// NETWORK 4
gvl_axis.fbi_mc_absR(
    Axis := gvl_axis.axisR,
    Execute := gvl_axis.ref_r.Execute,
    Position := gvl_axis.ref_r.Position,
    Velocity := gvl_axis.ref_r.Velocity,
    Acceleration := gvl_axis.ref_r.Acceleration,
    Deceleration := gvl_axis.ref_r.Deceleration,
    Jerk := gvl_axis.ref_r.Jerk,
    BufferMode := gvl_axis.ref_r.BufferMode,
    Options := gvl_axis.ref_r.Options,
    Busy => gvl_axis.ref_r.Busy,
    Active => gvl_axis.ref_r.Active,
    CommandAborted => gvl_axis.ref_r.CommandAborted,
    Error => gvl_axis.ref_r.Error,
    ErrorID => gvl_axis.ref_r.ErrorID); // MC_MoveAbsolute
gvl_axis.ref_r.Done := gvl_axis.fbi_mc_absR.Done;

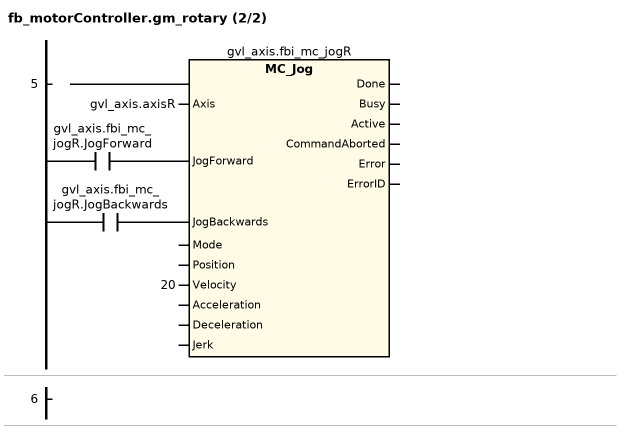
// NETWORK 5
gvl_axis.fbi_mc_jogR(
    Axis := gvl_axis.axisR,
    JogForward := gvl_axis.fbi_mc_jogR.JogForward,
    JogBackwards := gvl_axis.fbi_mc_jogR.JogBackwards,
    Velocity := 20); // MC_Jog

// NETWORK 6
END_ACTION

ACTION motorJog:
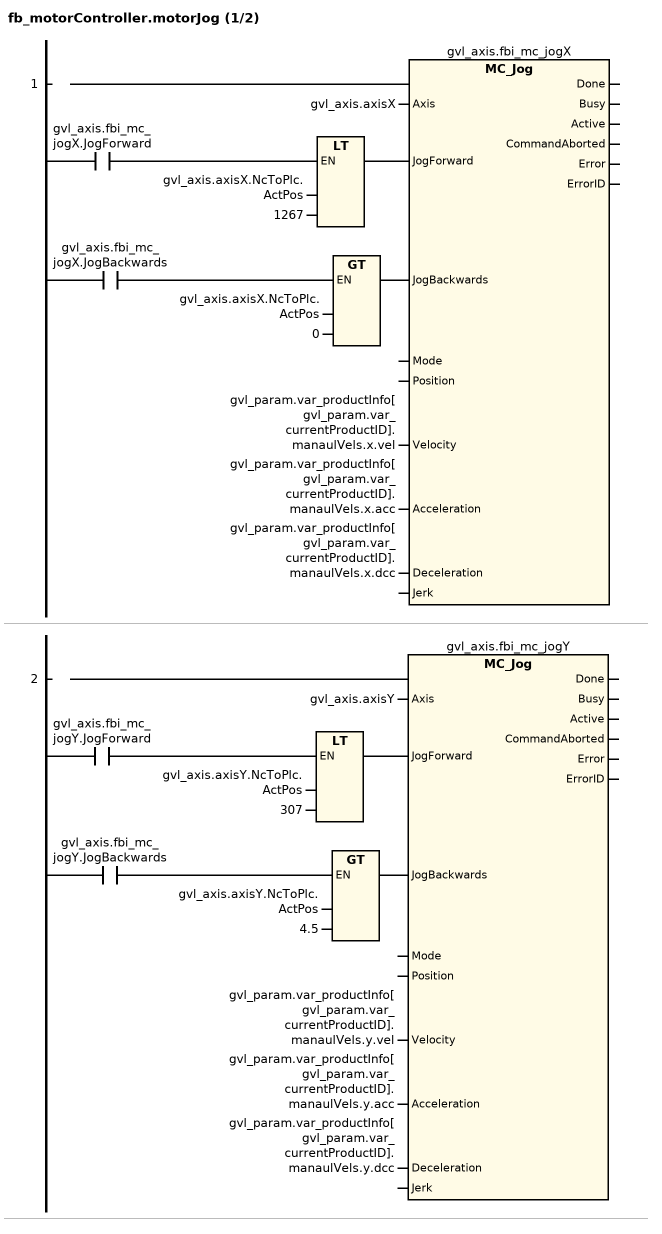
// NETWORK 1
gvl_axis.fbi_mc_jogX(
    Axis := gvl_axis.axisX,
    JogForward := gvl_axis.fbi_mc_jogX.JogForward AND gvl_axis.axisX.NcToPlc.ActPos < 1267,
    JogBackwards := gvl_axis.fbi_mc_jogX.JogBackwards AND gvl_axis.axisX.NcToPlc.ActPos > 0,
    Velocity := gvl_param.var_productInfo[gvl_param.var_currentProductID].manaulVels.x.vel,
    Acceleration := gvl_param.var_productInfo[gvl_param.var_currentProductID].manaulVels.x.acc,
    Deceleration := gvl_param.var_productInfo[gvl_param.var_currentProductID].manaulVels.x.dcc); // MC_Jog

// NETWORK 2
gvl_axis.fbi_mc_jogY(
    Axis := gvl_axis.axisY,
    JogForward := gvl_axis.fbi_mc_jogY.JogForward AND gvl_axis.axisY.NcToPlc.ActPos < 307,
    JogBackwards := gvl_axis.fbi_mc_jogY.JogBackwards AND gvl_axis.axisY.NcToPlc.ActPos > 4.5,
    Velocity := gvl_param.var_productInfo[gvl_param.var_currentProductID].manaulVels.y.vel,
    Acceleration := gvl_param.var_productInfo[gvl_param.var_currentProductID].manaulVels.y.acc,
    Deceleration := gvl_param.var_productInfo[gvl_param.var_currentProductID].manaulVels.y.dcc); // MC_Jog

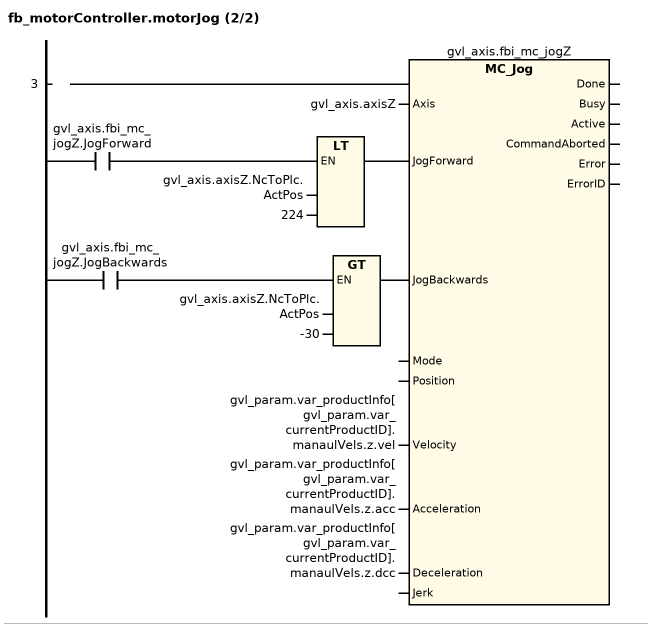
// NETWORK 3
gvl_axis.fbi_mc_jogZ(
    Axis := gvl_axis.axisZ,
    JogForward := gvl_axis.fbi_mc_jogZ.JogForward AND gvl_axis.axisZ.NcToPlc.ActPos < 224,
    JogBackwards := gvl_axis.fbi_mc_jogZ.JogBackwards AND gvl_axis.axisZ.NcToPlc.ActPos > -30,
    Velocity := gvl_param.var_productInfo[gvl_param.var_currentProductID].manaulVels.z.vel,
    Acceleration := gvl_param.var_productInfo[gvl_param.var_currentProductID].manaulVels.z.acc,
    Deceleration := gvl_param.var_productInfo[gvl_param.var_currentProductID].manaulVels.z.dcc); // MC_Jog
END_ACTION

ACTION motorMoveAbs:
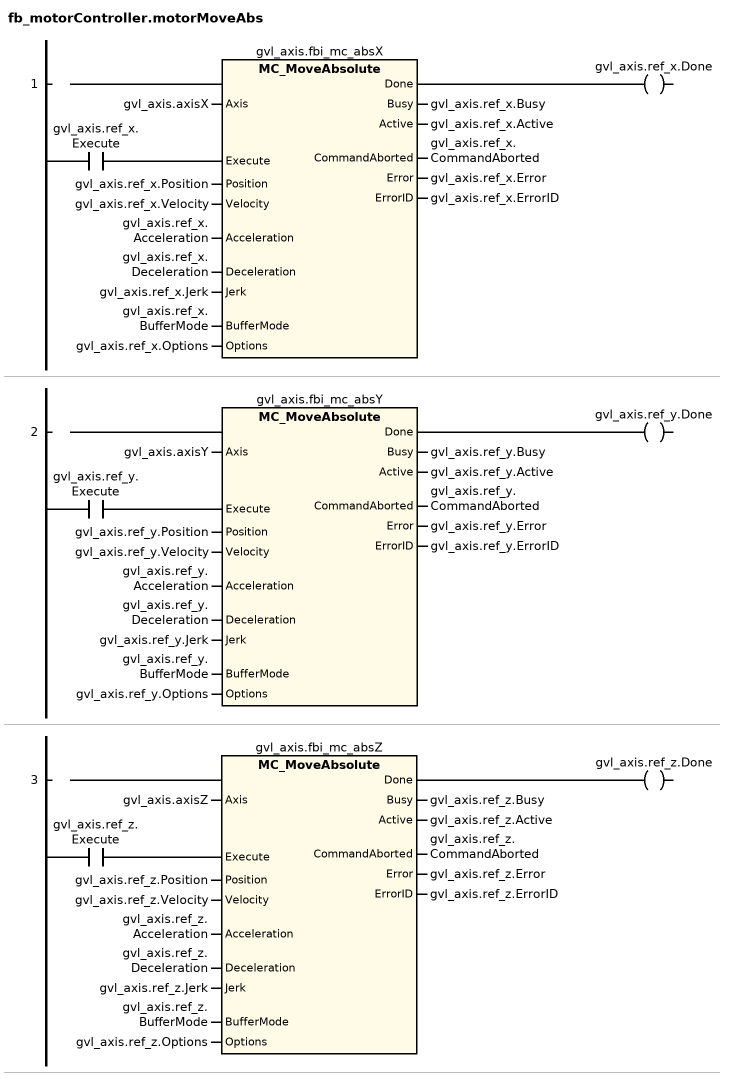
// NETWORK 1
gvl_axis.fbi_mc_absX(
    Axis := gvl_axis.axisX,
    Execute := gvl_axis.ref_x.Execute,
    Position := gvl_axis.ref_x.Position,
    Velocity := gvl_axis.ref_x.Velocity,
    Acceleration := gvl_axis.ref_x.Acceleration,
    Deceleration := gvl_axis.ref_x.Deceleration,
    Jerk := gvl_axis.ref_x.Jerk,
    BufferMode := gvl_axis.ref_x.BufferMode,
    Options := gvl_axis.ref_x.Options,
    Busy => gvl_axis.ref_x.Busy,
    Active => gvl_axis.ref_x.Active,
    CommandAborted => gvl_axis.ref_x.CommandAborted,
    Error => gvl_axis.ref_x.Error,
    ErrorID => gvl_axis.ref_x.ErrorID); // MC_MoveAbsolute
gvl_axis.ref_x.Done := gvl_axis.fbi_mc_absX.Done;

// NETWORK 2
gvl_axis.fbi_mc_absY(
    Axis := gvl_axis.axisY,
    Execute := gvl_axis.ref_y.Execute,
    Position := gvl_axis.ref_y.Position,
    Velocity := gvl_axis.ref_y.Velocity,
    Acceleration := gvl_axis.ref_y.Acceleration,
    Deceleration := gvl_axis.ref_y.Deceleration,
    Jerk := gvl_axis.ref_y.Jerk,
    BufferMode := gvl_axis.ref_y.BufferMode,
    Options := gvl_axis.ref_y.Options,
    Busy => gvl_axis.ref_y.Busy,
    Active => gvl_axis.ref_y.Active,
    CommandAborted => gvl_axis.ref_y.CommandAborted,
    Error => gvl_axis.ref_y.Error,
    ErrorID => gvl_axis.ref_y.ErrorID); // MC_MoveAbsolute
gvl_axis.ref_y.Done := gvl_axis.fbi_mc_absY.Done;

// NETWORK 3
gvl_axis.fbi_mc_absZ(
    Axis := gvl_axis.axisZ,
    Execute := gvl_axis.ref_z.Execute,
    Position := gvl_axis.ref_z.Position,
    Velocity := gvl_axis.ref_z.Velocity,
    Acceleration := gvl_axis.ref_z.Acceleration,
    Deceleration := gvl_axis.ref_z.Deceleration,
    Jerk := gvl_axis.ref_z.Jerk,
    BufferMode := gvl_axis.ref_z.BufferMode,
    Options := gvl_axis.ref_z.Options,
    Busy => gvl_axis.ref_z.Busy,
    Active => gvl_axis.ref_z.Active,
    CommandAborted => gvl_axis.ref_z.CommandAborted,
    Error => gvl_axis.ref_z.Error,
    ErrorID => gvl_axis.ref_z.ErrorID); // MC_MoveAbsolute
gvl_axis.ref_z.Done := gvl_axis.fbi_mc_absZ.Done;
END_ACTION

ACTION motorPower:
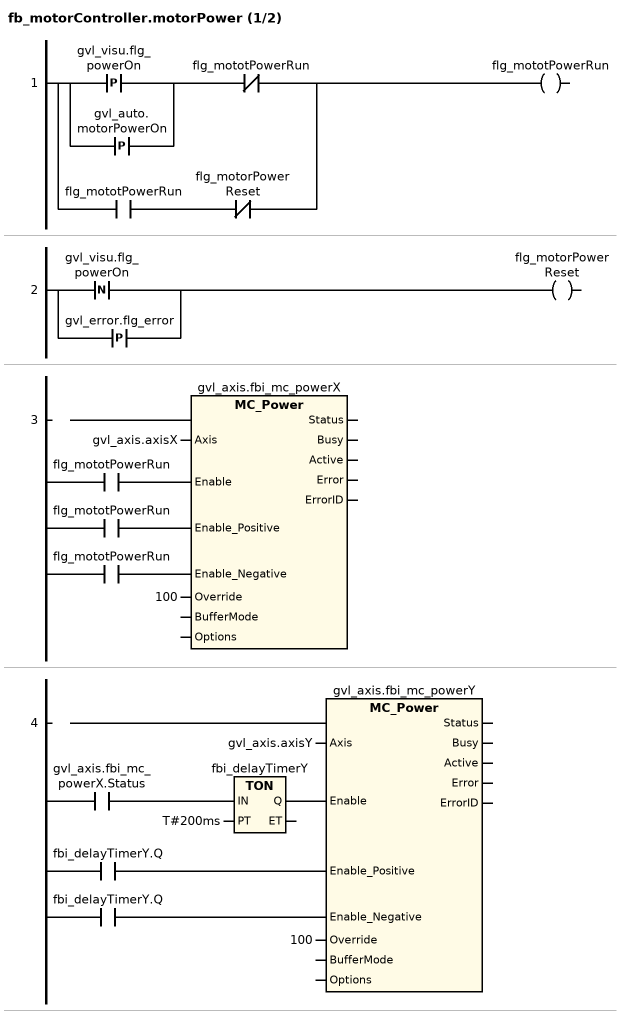
// NETWORK 1
_rt4(CLK := gvl_visu.flg_powerOn);
_rt5(CLK := gvl_auto.motorPowerOn);
flg_mototPowerRun := (_rt4.Q OR _rt5.Q) AND NOT flg_mototPowerRun OR flg_mototPowerRun AND NOT flg_motorPowerReset;

// NETWORK 2
_ft2(CLK := gvl_visu.flg_powerOn);
_rt6(CLK := gvl_error.flg_error);
flg_motorPowerReset := _ft2.Q OR _rt6.Q;

// NETWORK 3
gvl_axis.fbi_mc_powerX(
    Axis := gvl_axis.axisX,
    Enable := flg_mototPowerRun,
    Enable_Positive := flg_mototPowerRun,
    Enable_Negative := flg_mototPowerRun,
    Override := 100); // MC_Power

// NETWORK 4
fbi_delayTimerY(IN := gvl_axis.fbi_mc_powerX.Status, PT := T#200ms); // TON
gvl_axis.fbi_mc_powerY(
    Axis := gvl_axis.axisY,
    Enable := fbi_delayTimerY.Q,
    Enable_Positive := fbi_delayTimerY.Q,
    Enable_Negative := fbi_delayTimerY.Q,
    Override := 100); // MC_Power

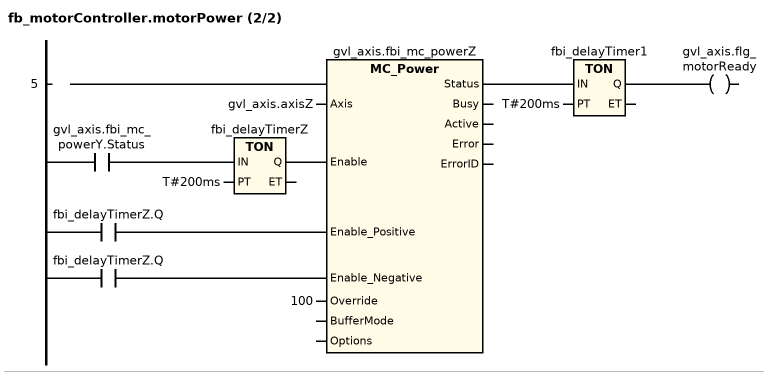
// NETWORK 5
fbi_delayTimerZ(IN := gvl_axis.fbi_mc_powerY.Status, PT := T#200ms); // TON
gvl_axis.fbi_mc_powerZ(
    Axis := gvl_axis.axisZ,
    Enable := fbi_delayTimerZ.Q,
    Enable_Positive := fbi_delayTimerZ.Q,
    Enable_Negative := fbi_delayTimerZ.Q,
    Override := 100); // MC_Power
fbi_delayTimer1(IN := gvl_axis.fbi_mc_powerZ.Status, PT := T#200ms); // TON
gvl_axis.flg_motorReady := fbi_delayTimer1.Q;
END_ACTION

END_FUNCTION_BLOCK

// ---- FBs/error/fb_eventController.TcPOU
FUNCTION_BLOCK fb_eventController
VAR_INPUT
in_flg_run : BOOL;
END_VAR
VAR_OUTPUT
	out_flg_run : BOOL;
END_VAR
VAR

	fbi_eventListGenerator: ARRAY [0..50] OF fb_eventListGenerator;
	var_semaphore: INT;
	var_alarmQty: INT;
	flg_errorTrg: ARRAY[0..50] OF BOOL;

    var_timeAsDT : DT;
	var_alarmListLog: s_alarmList;
	flg_reqUpdate: BOOL;
	fbi_r_TRIG: R_TRIG;
	var_n: INT;
	fbi_buzzerGenerater: fb_buzzerGenerater;
	var_n2: INT;
	var_alarmListEmpty : s_alarmList;
	fbi_GetLocalAmsNetId: FB_GetLocalAmsNetId;
	fbi_LocalSystemTime: FB_LocalSystemTime;
	fbi_ton1: TON;
	var_i: INT;
	fbi_first: TON;
	var_dummy: ARRAY [1..10] OF s_str_alarmList;
END_VAR
VAR_STAT
	flg_error: BOOL;
	flg_warning: BOOL;
	flg_info: BOOL;
END_VAR
VAR // added by the converter: edge detectors and wires of the graphical bodies
    _rt1 : R_TRIG;
END_VAR

eventList();

//get current time
fbi_GetLocalAmsNetId(
	bExecute:=TRUE , 
	tTimeOut:= ,
	bBusy=> , 
	bError=> , 
	nErrId=> , 
	AddrString=> , 
	AddrBytes=> );


fbi_LocalSystemTime(
	sNetID:=fbi_GetLocalAmsNetId.AddrString , 
	bEnable:= TRUE, 
	dwCycle:= , 
	dwOpt:= , 
	tTimeout:= , 
	bValid=> , 
	systemTime=> , 
	tzID=> );

var_timeAsDT := SYSTEMTIME_TO_DT(fbi_LocalSystemTime.systemTime);
//reset

//
IF gvl_error.flg_error THEN
	gvl_error.flg_alramBusy := TRUE;
END_IF

fbi_r_TRIG(CLK:= flg_requpdate, Q=> );
//event log update
IF fbi_r_TRIG.Q THEN
	FOR var_n := 50 TO 2 BY -1 DO
			gvl_error.var_ary_alarmlistLog[var_n].var_alarmName := gvl_error.var_ary_alarmlistLog[var_n-1].var_alarmName;
			gvl_error.var_ary_alarmlistLog[var_n].var_alarmLevel := gvl_error.var_ary_alarmlistLog[var_n-1].var_alarmLevel;
			gvl_error.var_ary_alarmlistLog[var_n].var_alarmMassge := gvl_error.var_ary_alarmlistLog[var_n-1].var_alarmMassge;
			gvl_error.var_ary_alarmlistLog[var_n].var_alarmTime := gvl_error.var_ary_alarmlistLog[var_n-1].var_alarmTime;
			gvl_error.var_ary_alarmlistLog[var_n].var_alarmCode1 := gvl_error.var_ary_alarmlistLog[var_n-1].var_alarmCode1;
			gvl_error.var_ary_alarmlistLog[var_n].var_alarmCode2 := gvl_error.var_ary_alarmlistLog[var_n-1].var_alarmCode2;
			
			IF var_n = 2 THEN
				gvl_error.var_ary_alarmlistLog[1].var_alarmName := var_alarmListLog.var_alarmName;
				gvl_error.var_ary_alarmlistLog[1].var_alarmLevel := var_alarmListLog.var_alarmLevel;
				gvl_error.var_ary_alarmlistLog[1].var_alarmMassge := var_alarmListLog.var_alarmMassge;
				gvl_error.var_ary_alarmlistLog[1].var_alarmTime := var_alarmListLog.var_alarmTime;
				gvl_error.var_ary_alarmlistLog[1].var_alarmCode1 := var_alarmListLog.var_alarmCode1;
				gvl_error.var_ary_alarmlistLog[1].var_alarmCode2 := var_alarmListLog.var_alarmCode2;
				var_semaphore := var_semaphore - 1;
			END_IF
		END_FOR	
END_IF

//reset realtime event 
IF gvl_error.flg_eventDisplayRest THEN
	FOR var_n2 := 1 TO 10 BY 1 DO
		gvl_error.var_ary_alarmlistActive[var_n2].var_alarmCode1 := eP_alarmCode._;
		gvl_error.var_ary_alarmlistActive[var_n2].var_alarmCode2 := '';
		gvl_error.var_ary_alarmlistActive[var_n2].var_alarmLevel := '';
		gvl_error.var_ary_alarmlistActive[var_n2].var_alarmMassge := "";
		gvl_error.var_ary_alarmlistActive[var_n2].var_alarmName := "";
		gvl_error.var_ary_alarmlistActive[var_n2].var_alarmTime := '';
	END_FOR
END_IF
//massage
	flg_info := gvl_error.flg_warning OR gvl_error.flg_info OR gvl_error.flg_sample_windown_warning;
	IF NOT flg_info THEN
		gvl_visu.var_msg := "";	
	END_IF
//buzzer
fbi_buzzerGenerater(
	in_flg_LvError:=gvl_error.flg_error OR gvl_error.flg_sample_windown_warning,
	in_flg_LvWarning:=gvl_error.flg_warning,
	in_flg_LvInfo:=gvl_error.flg_info ,
	out_flg_buzzer=> gvl_io.flg_signalTowerBuzzer ,
	out_flg_Yellow=> gvl_io.flg_signalTowerYellow
);
gvl_io.flg_signalTowerRed := gvl_error.flg_error;

IF gvl_error.flg_ararmLevelRest THEN
	gvl_error.flg_error := FALSE;
	gvl_error.flg_warning := FALSE;
	gvl_error.flg_info := FALSE;
END_IF

ACTION eventList:
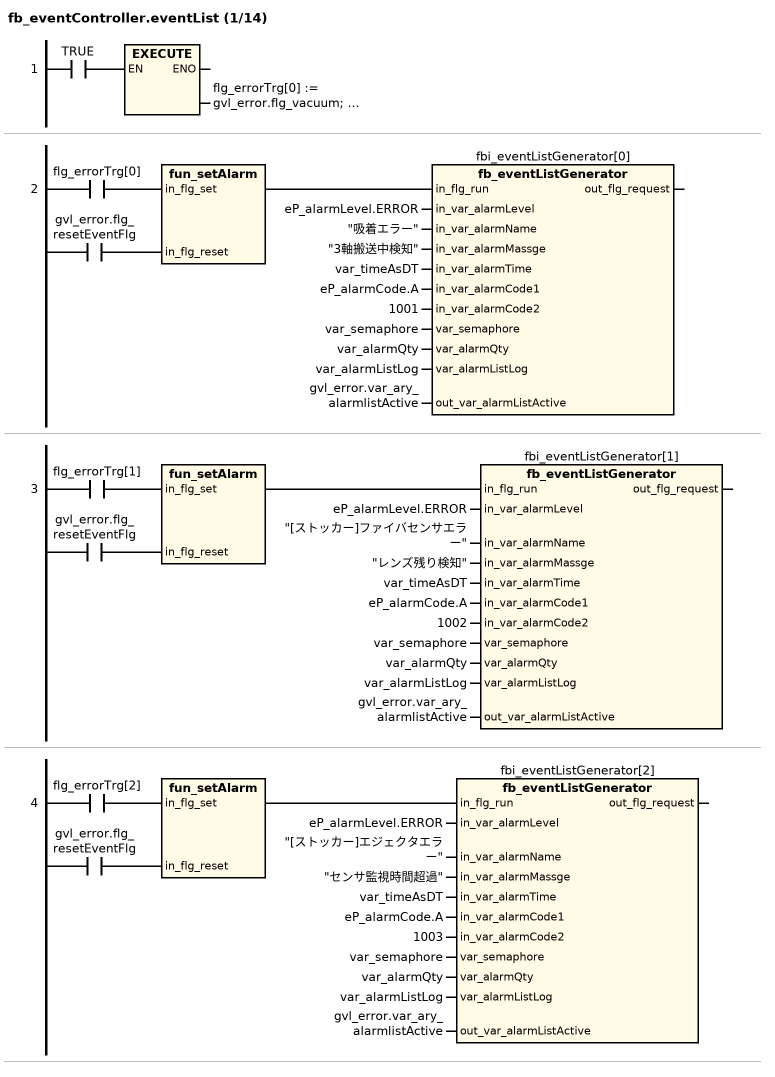
// NETWORK 1
flg_errorTrg[0] := gvl_error.flg_vacuum;
flg_errorTrg[1] := gvl_error.flg_fiberSens;
flg_errorTrg[2] := gvl_solv.fbi_ejector.out_flg_error;
flg_errorTrg[3] := gvl_solv.fbi_chuck.out_flg_error;
flg_errorTrg[4] := gvl_solv.fbi_push.out_flg_error;
flg_errorTrg[5] := gvl_elecylinder.fbi_axisTransport.out_flg_error;
flg_errorTrg[6] := gvl_elecylinder.fbi_axisSample.out_flg_error;
flg_errorTrg[7] := gvl_elecylinder.fbi_axisTrayChange.out_flg_error OR gvl_error.flg_trayChangeError;
flg_errorTrg[8] := gvl_elecylinder.ref_axis_transport.input.in_wire_error;
flg_errorTrg[9] := gvl_elecylinder.ref_axis_sample.input.in_wire_error;
flg_errorTrg[10] := gvl_elecylinder.ref_axis_trayChange.input.in_wire_error;
flg_errorTrg[11] := gvl_axis.ref_x.Error;
flg_errorTrg[12] := gvl_axis.ref_y.Error;
flg_errorTrg[13] := gvl_axis.ref_z.Error;
flg_errorTrg[14] := gvl_elecylinder.fbi_axisRotary.out_flg_error;
flg_errorTrg[15] := gvl_elecylinder.ref_axis_rotary.input.in_wire_error;
flg_errorTrg[16] := NOT gvl_io.flg_saftyUnitState;
flg_errorTrg[17] := NOT gvl_io.flg_frontSaftyDoor;
flg_errorTrg[18] := gvl_io.flg_gatemeasurementStatus;
flg_errorTrg[19] := gvl_axis.fbi_mc_jogX.Error;
flg_errorTrg[20] := gvl_axis.fbi_mc_jogY.Error;
flg_errorTrg[21] := gvl_axis.fbi_mc_jogZ.Error;
flg_errorTrg[22] := gvl_auto.flg_trayChangeDone OR NOT  gvl_visu.flg_btn_trayChangeDone ;
flg_errorTrg[23] := gvl_error.flg_gm_fiberSens; 
flg_errorTrg[24] := gvl_solv.fbi_gm_ejector.out_flg_error;
flg_errorTrg[25] := gvl_solv.fbi_gm_chuck.out_flg_error;
flg_errorTrg[26] := gvl_solv.fbi_gm_push.out_flg_error;
flg_errorTrg[27] := gvl_elecylinder.fbi_gm_axisPickUp.out_flg_error;
flg_errorTrg[28] := gvl_elecylinder.fbi_gm_axisTransport.out_flg_error;
flg_errorTrg[29] := gvl_axis.ref_r.Error;
flg_errorTrg[30] := gvl_axis.fbi_mc_jogR.Error;
flg_errorTrg[31] := gvl_error.flg_axisXTorqueOver;
flg_errorTrg[32] := gvl_error.flg_axisYTorqueOver;
flg_errorTrg[33] := gvl_error.flg_axisZTorqueOver;
flg_errorTrg[34] := gvl_error.flg_axisRTorqueOver;
flg_errorTrg[35] := gvl_solv.fbi_gm_rotary.out_flg_error;
flg_errorTrg[36] := gvl_solv.fbi_gm_pickup.out_flg_error;
flg_errorTrg[37] := gvl_solv.fbi_gm_stamp.out_flg_error;
flg_errorTrg[38] := gvl_gm.var_incjetInfo.flg_error;
flg_errorTrg[39] := gvl_error.flg_incjet;
flg_errorTrg[40] := gvl_error.flg_sample_windown_error;
//flg_errorTrg[41] := ;
//flg_errorTrg[42] := ;
//flg_errorTrg[43] := ;
//flg_errorTrg[44] := ;
//flg_errorTrg[45] := ;
//flg_errorTrg[46] := ;
//flg_errorTrg[47] := ;
//flg_errorTrg[48] := ;
//flg_errorTrg[49] := ;
//flg_errorTrg[50] := ;

// NETWORK 2
fbi_eventListGenerator[0](
    in_flg_run := fun_setAlarm(in_flg_set := flg_errorTrg[0], in_flg_reset := gvl_error.flg_resetEventFlg),
    in_var_alarmLevel := eP_alarmLevel.ERROR,
    in_var_alarmName := "吸着エラー",
    in_var_alarmMassge := "3軸搬送中検知",
    in_var_alarmTime := var_timeAsDT,
    in_var_alarmCode1 := eP_alarmCode.A,
    in_var_alarmCode2 := 1001,
    var_semaphore := var_semaphore,
    var_alarmQty := var_alarmQty,
    var_alarmListLog := var_alarmListLog,
    out_var_alarmListActive := gvl_error.var_ary_alarmlistActive); // fb_eventListGenerator

// NETWORK 3
fbi_eventListGenerator[1](
    in_flg_run := fun_setAlarm(in_flg_set := flg_errorTrg[1], in_flg_reset := gvl_error.flg_resetEventFlg),
    in_var_alarmLevel := eP_alarmLevel.ERROR,
    in_var_alarmName := "[ストッカー]ファイバセンサエラー",
    in_var_alarmMassge := "レンズ残り検知",
    in_var_alarmTime := var_timeAsDT,
    in_var_alarmCode1 := eP_alarmCode.A,
    in_var_alarmCode2 := 1002,
    var_semaphore := var_semaphore,
    var_alarmQty := var_alarmQty,
    var_alarmListLog := var_alarmListLog,
    out_var_alarmListActive := gvl_error.var_ary_alarmlistActive); // fb_eventListGenerator

// NETWORK 4
fbi_eventListGenerator[2](
    in_flg_run := fun_setAlarm(in_flg_set := flg_errorTrg[2], in_flg_reset := gvl_error.flg_resetEventFlg),
    in_var_alarmLevel := eP_alarmLevel.ERROR,
    in_var_alarmName := "[ストッカー]エジェクタエラー",
    in_var_alarmMassge := "センサ監視時間超過",
    in_var_alarmTime := var_timeAsDT,
    in_var_alarmCode1 := eP_alarmCode.A,
    in_var_alarmCode2 := 1003,
    var_semaphore := var_semaphore,
    var_alarmQty := var_alarmQty,
    var_alarmListLog := var_alarmListLog,
    out_var_alarmListActive := gvl_error.var_ary_alarmlistActive); // fb_eventListGenerator

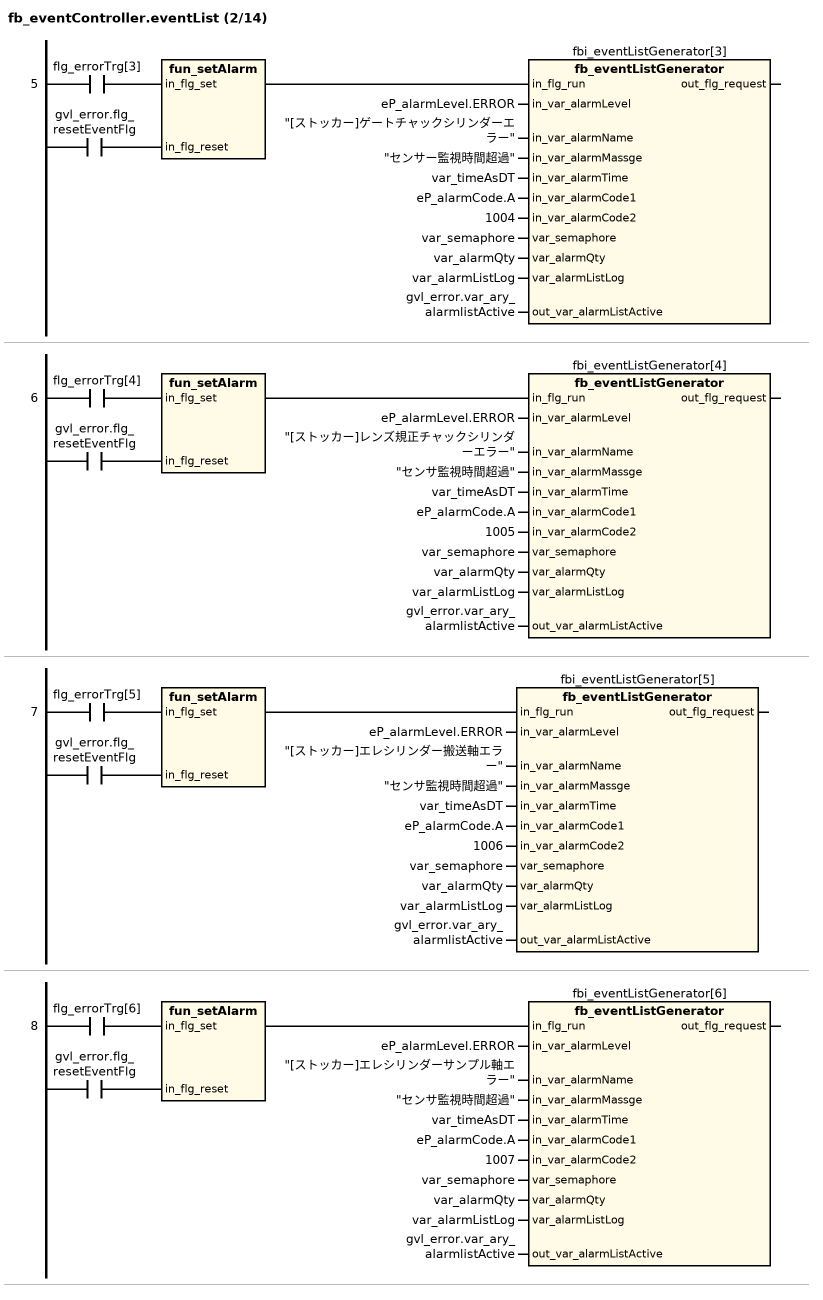
// NETWORK 5
fbi_eventListGenerator[3](
    in_flg_run := fun_setAlarm(in_flg_set := flg_errorTrg[3], in_flg_reset := gvl_error.flg_resetEventFlg),
    in_var_alarmLevel := eP_alarmLevel.ERROR,
    in_var_alarmName := "[ストッカー]ゲートチャックシリンダーエラー",
    in_var_alarmMassge := "センサー監視時間超過",
    in_var_alarmTime := var_timeAsDT,
    in_var_alarmCode1 := eP_alarmCode.A,
    in_var_alarmCode2 := 1004,
    var_semaphore := var_semaphore,
    var_alarmQty := var_alarmQty,
    var_alarmListLog := var_alarmListLog,
    out_var_alarmListActive := gvl_error.var_ary_alarmlistActive); // fb_eventListGenerator

// NETWORK 6
fbi_eventListGenerator[4](
    in_flg_run := fun_setAlarm(in_flg_set := flg_errorTrg[4], in_flg_reset := gvl_error.flg_resetEventFlg),
    in_var_alarmLevel := eP_alarmLevel.ERROR,
    in_var_alarmName := "[ストッカー]レンズ規正チャックシリンダーエラー",
    in_var_alarmMassge := "センサ監視時間超過",
    in_var_alarmTime := var_timeAsDT,
    in_var_alarmCode1 := eP_alarmCode.A,
    in_var_alarmCode2 := 1005,
    var_semaphore := var_semaphore,
    var_alarmQty := var_alarmQty,
    var_alarmListLog := var_alarmListLog,
    out_var_alarmListActive := gvl_error.var_ary_alarmlistActive); // fb_eventListGenerator

// NETWORK 7
fbi_eventListGenerator[5](
    in_flg_run := fun_setAlarm(in_flg_set := flg_errorTrg[5], in_flg_reset := gvl_error.flg_resetEventFlg),
    in_var_alarmLevel := eP_alarmLevel.ERROR,
    in_var_alarmName := "[ストッカー]エレシリンダー搬送軸エラー",
    in_var_alarmMassge := "センサ監視時間超過",
    in_var_alarmTime := var_timeAsDT,
    in_var_alarmCode1 := eP_alarmCode.A,
    in_var_alarmCode2 := 1006,
    var_semaphore := var_semaphore,
    var_alarmQty := var_alarmQty,
    var_alarmListLog := var_alarmListLog,
    out_var_alarmListActive := gvl_error.var_ary_alarmlistActive); // fb_eventListGenerator

// NETWORK 8
fbi_eventListGenerator[6](
    in_flg_run := fun_setAlarm(in_flg_set := flg_errorTrg[6], in_flg_reset := gvl_error.flg_resetEventFlg),
    in_var_alarmLevel := eP_alarmLevel.ERROR,
    in_var_alarmName := "[ストッカー]エレシリンダーサンプル軸エラー",
    in_var_alarmMassge := "センサ監視時間超過",
    in_var_alarmTime := var_timeAsDT,
    in_var_alarmCode1 := eP_alarmCode.A,
    in_var_alarmCode2 := 1007,
    var_semaphore := var_semaphore,
    var_alarmQty := var_alarmQty,
    var_alarmListLog := var_alarmListLog,
    out_var_alarmListActive := gvl_error.var_ary_alarmlistActive); // fb_eventListGenerator

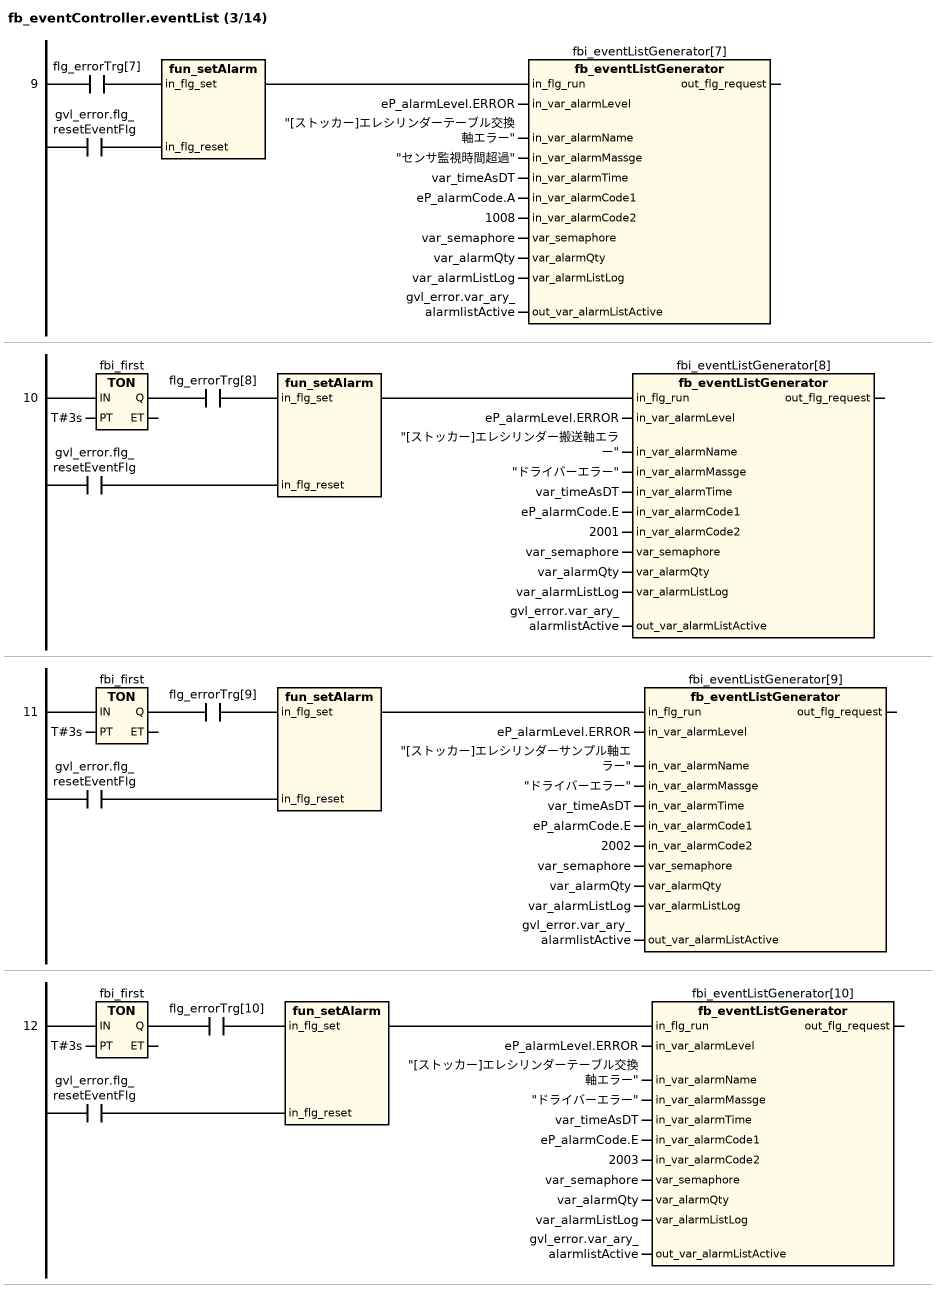
// NETWORK 9
fbi_eventListGenerator[7](
    in_flg_run := fun_setAlarm(in_flg_set := flg_errorTrg[7], in_flg_reset := gvl_error.flg_resetEventFlg),
    in_var_alarmLevel := eP_alarmLevel.ERROR,
    in_var_alarmName := "[ストッカー]エレシリンダーテーブル交換軸エラー",
    in_var_alarmMassge := "センサ監視時間超過",
    in_var_alarmTime := var_timeAsDT,
    in_var_alarmCode1 := eP_alarmCode.A,
    in_var_alarmCode2 := 1008,
    var_semaphore := var_semaphore,
    var_alarmQty := var_alarmQty,
    var_alarmListLog := var_alarmListLog,
    out_var_alarmListActive := gvl_error.var_ary_alarmlistActive); // fb_eventListGenerator

// NETWORK 10
fbi_first(IN := TRUE, PT := T#3s); // TON
fbi_eventListGenerator[8](
    in_flg_run := fun_setAlarm(in_flg_set := fbi_first.Q AND flg_errorTrg[8], in_flg_reset := gvl_error.flg_resetEventFlg),
    in_var_alarmLevel := eP_alarmLevel.ERROR,
    in_var_alarmName := "[ストッカー]エレシリンダー搬送軸エラー",
    in_var_alarmMassge := "ドライバーエラー",
    in_var_alarmTime := var_timeAsDT,
    in_var_alarmCode1 := eP_alarmCode.E,
    in_var_alarmCode2 := 2001,
    var_semaphore := var_semaphore,
    var_alarmQty := var_alarmQty,
    var_alarmListLog := var_alarmListLog,
    out_var_alarmListActive := gvl_error.var_ary_alarmlistActive); // fb_eventListGenerator

// NETWORK 11
fbi_first(IN := TRUE, PT := T#3s); // TON
fbi_eventListGenerator[9](
    in_flg_run := fun_setAlarm(in_flg_set := fbi_first.Q AND flg_errorTrg[9], in_flg_reset := gvl_error.flg_resetEventFlg),
    in_var_alarmLevel := eP_alarmLevel.ERROR,
    in_var_alarmName := "[ストッカー]エレシリンダーサンプル軸エラー",
    in_var_alarmMassge := "ドライバーエラー",
    in_var_alarmTime := var_timeAsDT,
    in_var_alarmCode1 := eP_alarmCode.E,
    in_var_alarmCode2 := 2002,
    var_semaphore := var_semaphore,
    var_alarmQty := var_alarmQty,
    var_alarmListLog := var_alarmListLog,
    out_var_alarmListActive := gvl_error.var_ary_alarmlistActive); // fb_eventListGenerator

// NETWORK 12
fbi_first(IN := TRUE, PT := T#3s); // TON
fbi_eventListGenerator[10](
    in_flg_run := fun_setAlarm(in_flg_set := fbi_first.Q AND flg_errorTrg[10], in_flg_reset := gvl_error.flg_resetEventFlg),
    in_var_alarmLevel := eP_alarmLevel.ERROR,
    in_var_alarmName := "[ストッカー]エレシリンダーテーブル交換軸エラー",
    in_var_alarmMassge := "ドライバーエラー",
    in_var_alarmTime := var_timeAsDT,
    in_var_alarmCode1 := eP_alarmCode.E,
    in_var_alarmCode2 := 2003,
    var_semaphore := var_semaphore,
    var_alarmQty := var_alarmQty,
    var_alarmListLog := var_alarmListLog,
    out_var_alarmListActive := gvl_error.var_ary_alarmlistActive); // fb_eventListGenerator

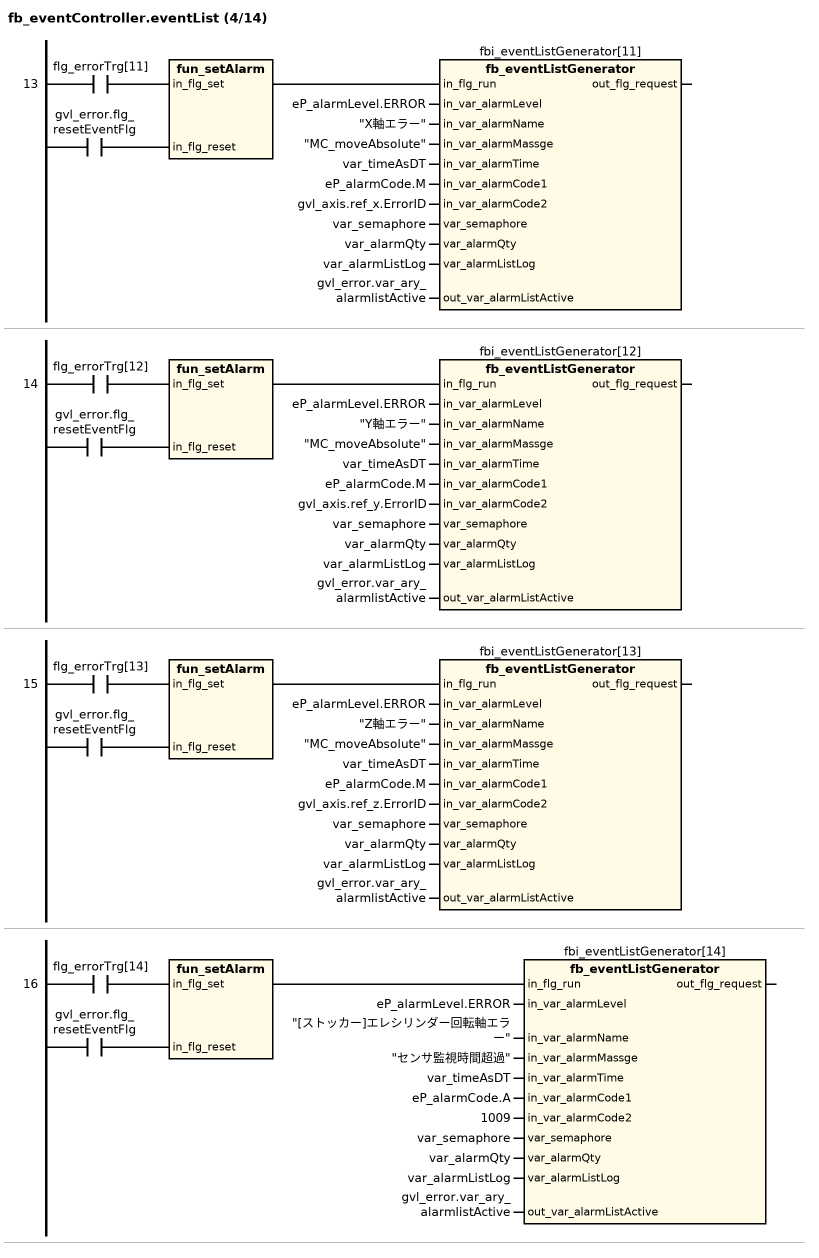
// NETWORK 13
fbi_eventListGenerator[11](
    in_flg_run := fun_setAlarm(in_flg_set := flg_errorTrg[11], in_flg_reset := gvl_error.flg_resetEventFlg),
    in_var_alarmLevel := eP_alarmLevel.ERROR,
    in_var_alarmName := "X軸エラー",
    in_var_alarmMassge := "MC_moveAbsolute",
    in_var_alarmTime := var_timeAsDT,
    in_var_alarmCode1 := eP_alarmCode.M,
    in_var_alarmCode2 := gvl_axis.ref_x.ErrorID,
    var_semaphore := var_semaphore,
    var_alarmQty := var_alarmQty,
    var_alarmListLog := var_alarmListLog,
    out_var_alarmListActive := gvl_error.var_ary_alarmlistActive); // fb_eventListGenerator

// NETWORK 14
fbi_eventListGenerator[12](
    in_flg_run := fun_setAlarm(in_flg_set := flg_errorTrg[12], in_flg_reset := gvl_error.flg_resetEventFlg),
    in_var_alarmLevel := eP_alarmLevel.ERROR,
    in_var_alarmName := "Y軸エラー",
    in_var_alarmMassge := "MC_moveAbsolute",
    in_var_alarmTime := var_timeAsDT,
    in_var_alarmCode1 := eP_alarmCode.M,
    in_var_alarmCode2 := gvl_axis.ref_y.ErrorID,
    var_semaphore := var_semaphore,
    var_alarmQty := var_alarmQty,
    var_alarmListLog := var_alarmListLog,
    out_var_alarmListActive := gvl_error.var_ary_alarmlistActive); // fb_eventListGenerator

// NETWORK 15
fbi_eventListGenerator[13](
    in_flg_run := fun_setAlarm(in_flg_set := flg_errorTrg[13], in_flg_reset := gvl_error.flg_resetEventFlg),
    in_var_alarmLevel := eP_alarmLevel.ERROR,
    in_var_alarmName := "Z軸エラー",
    in_var_alarmMassge := "MC_moveAbsolute",
    in_var_alarmTime := var_timeAsDT,
    in_var_alarmCode1 := eP_alarmCode.M,
    in_var_alarmCode2 := gvl_axis.ref_z.ErrorID,
    var_semaphore := var_semaphore,
    var_alarmQty := var_alarmQty,
    var_alarmListLog := var_alarmListLog,
    out_var_alarmListActive := gvl_error.var_ary_alarmlistActive); // fb_eventListGenerator

// NETWORK 16
fbi_eventListGenerator[14](
    in_flg_run := fun_setAlarm(in_flg_set := flg_errorTrg[14], in_flg_reset := gvl_error.flg_resetEventFlg),
    in_var_alarmLevel := eP_alarmLevel.ERROR,
    in_var_alarmName := "[ストッカー]エレシリンダー回転軸エラー",
    in_var_alarmMassge := "センサ監視時間超過",
    in_var_alarmTime := var_timeAsDT,
    in_var_alarmCode1 := eP_alarmCode.A,
    in_var_alarmCode2 := 1009,
    var_semaphore := var_semaphore,
    var_alarmQty := var_alarmQty,
    var_alarmListLog := var_alarmListLog,
    out_var_alarmListActive := gvl_error.var_ary_alarmlistActive); // fb_eventListGenerator

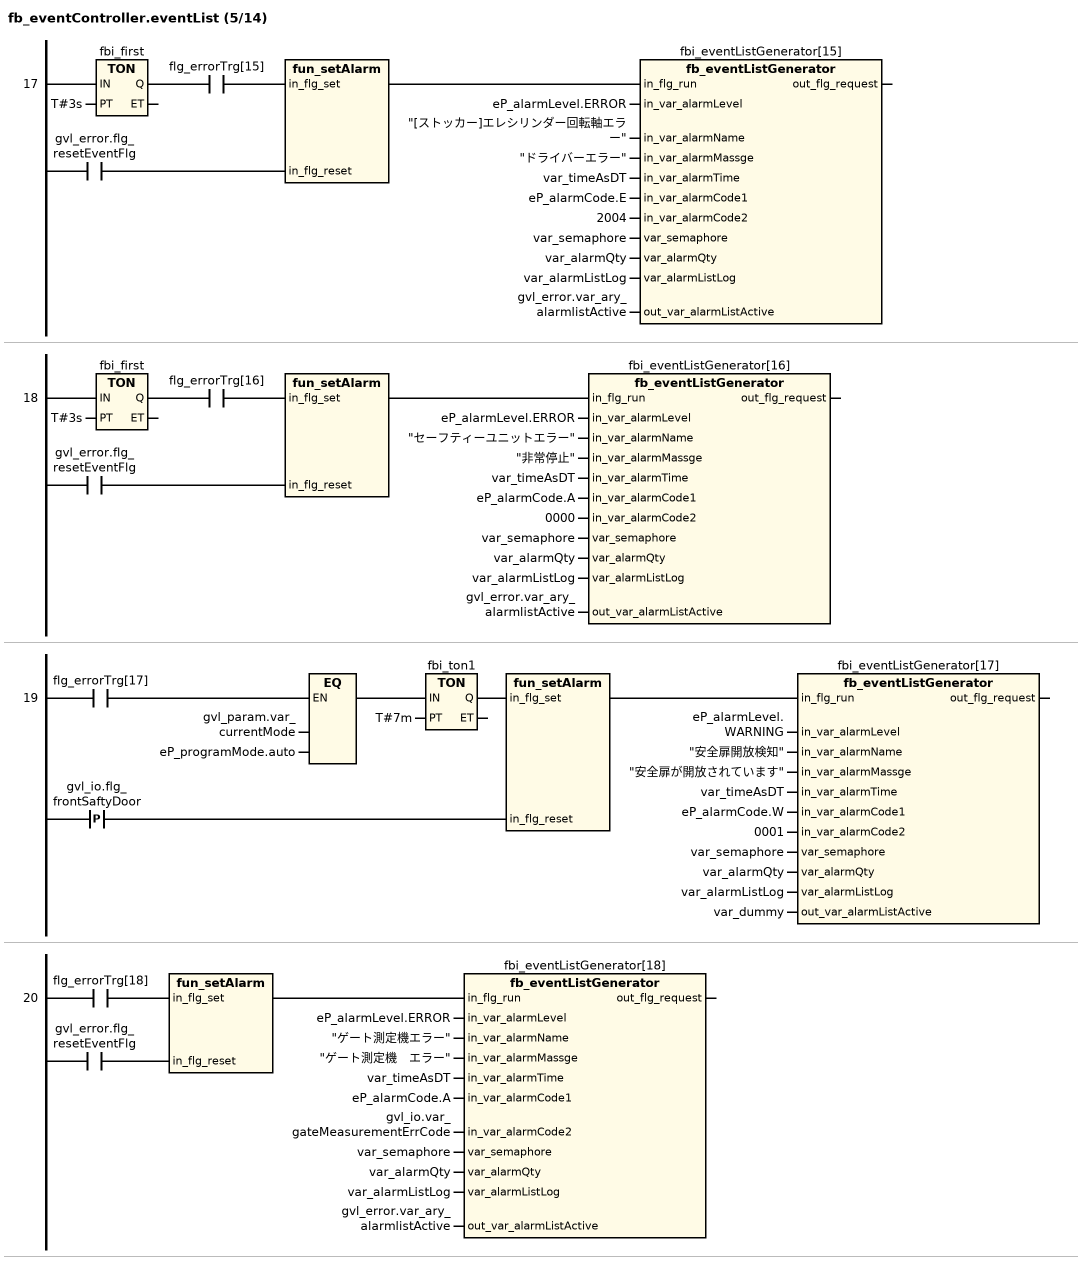
// NETWORK 17
fbi_first(IN := TRUE, PT := T#3s); // TON
fbi_eventListGenerator[15](
    in_flg_run := fun_setAlarm(in_flg_set := fbi_first.Q AND flg_errorTrg[15], in_flg_reset := gvl_error.flg_resetEventFlg),
    in_var_alarmLevel := eP_alarmLevel.ERROR,
    in_var_alarmName := "[ストッカー]エレシリンダー回転軸エラー",
    in_var_alarmMassge := "ドライバーエラー",
    in_var_alarmTime := var_timeAsDT,
    in_var_alarmCode1 := eP_alarmCode.E,
    in_var_alarmCode2 := 2004,
    var_semaphore := var_semaphore,
    var_alarmQty := var_alarmQty,
    var_alarmListLog := var_alarmListLog,
    out_var_alarmListActive := gvl_error.var_ary_alarmlistActive); // fb_eventListGenerator

// NETWORK 18
fbi_first(IN := TRUE, PT := T#3s); // TON
fbi_eventListGenerator[16](
    in_flg_run := fun_setAlarm(in_flg_set := fbi_first.Q AND flg_errorTrg[16], in_flg_reset := gvl_error.flg_resetEventFlg),
    in_var_alarmLevel := eP_alarmLevel.ERROR,
    in_var_alarmName := "セーフティーユニットエラー",
    in_var_alarmMassge := "非常停止",
    in_var_alarmTime := var_timeAsDT,
    in_var_alarmCode1 := eP_alarmCode.A,
    in_var_alarmCode2 := 0000,
    var_semaphore := var_semaphore,
    var_alarmQty := var_alarmQty,
    var_alarmListLog := var_alarmListLog,
    out_var_alarmListActive := gvl_error.var_ary_alarmlistActive); // fb_eventListGenerator

// NETWORK 19
fbi_ton1(IN := flg_errorTrg[17] AND gvl_param.var_currentMode = eP_programMode.auto, PT := T#7m); // TON
_rt1(CLK := gvl_io.flg_frontSaftyDoor);
fbi_eventListGenerator[17](
    in_flg_run := fun_setAlarm(in_flg_set := fbi_ton1.Q, in_flg_reset := _rt1.Q),
    in_var_alarmLevel := eP_alarmLevel.WARNING,
    in_var_alarmName := "安全扉開放検知",
    in_var_alarmMassge := "安全扉が開放されています",
    in_var_alarmTime := var_timeAsDT,
    in_var_alarmCode1 := eP_alarmCode.W,
    in_var_alarmCode2 := 0001,
    var_semaphore := var_semaphore,
    var_alarmQty := var_alarmQty,
    var_alarmListLog := var_alarmListLog,
    out_var_alarmListActive := var_dummy); // fb_eventListGenerator

// NETWORK 20
fbi_eventListGenerator[18](
    in_flg_run := fun_setAlarm(in_flg_set := flg_errorTrg[18], in_flg_reset := gvl_error.flg_resetEventFlg),
    in_var_alarmLevel := eP_alarmLevel.ERROR,
    in_var_alarmName := "ゲート測定機エラー",
    in_var_alarmMassge := "ゲート測定機　エラー",
    in_var_alarmTime := var_timeAsDT,
    in_var_alarmCode1 := eP_alarmCode.A,
    in_var_alarmCode2 := gvl_io.var_gateMeasurementErrCode,
    var_semaphore := var_semaphore,
    var_alarmQty := var_alarmQty,
    var_alarmListLog := var_alarmListLog,
    out_var_alarmListActive := gvl_error.var_ary_alarmlistActive); // fb_eventListGenerator

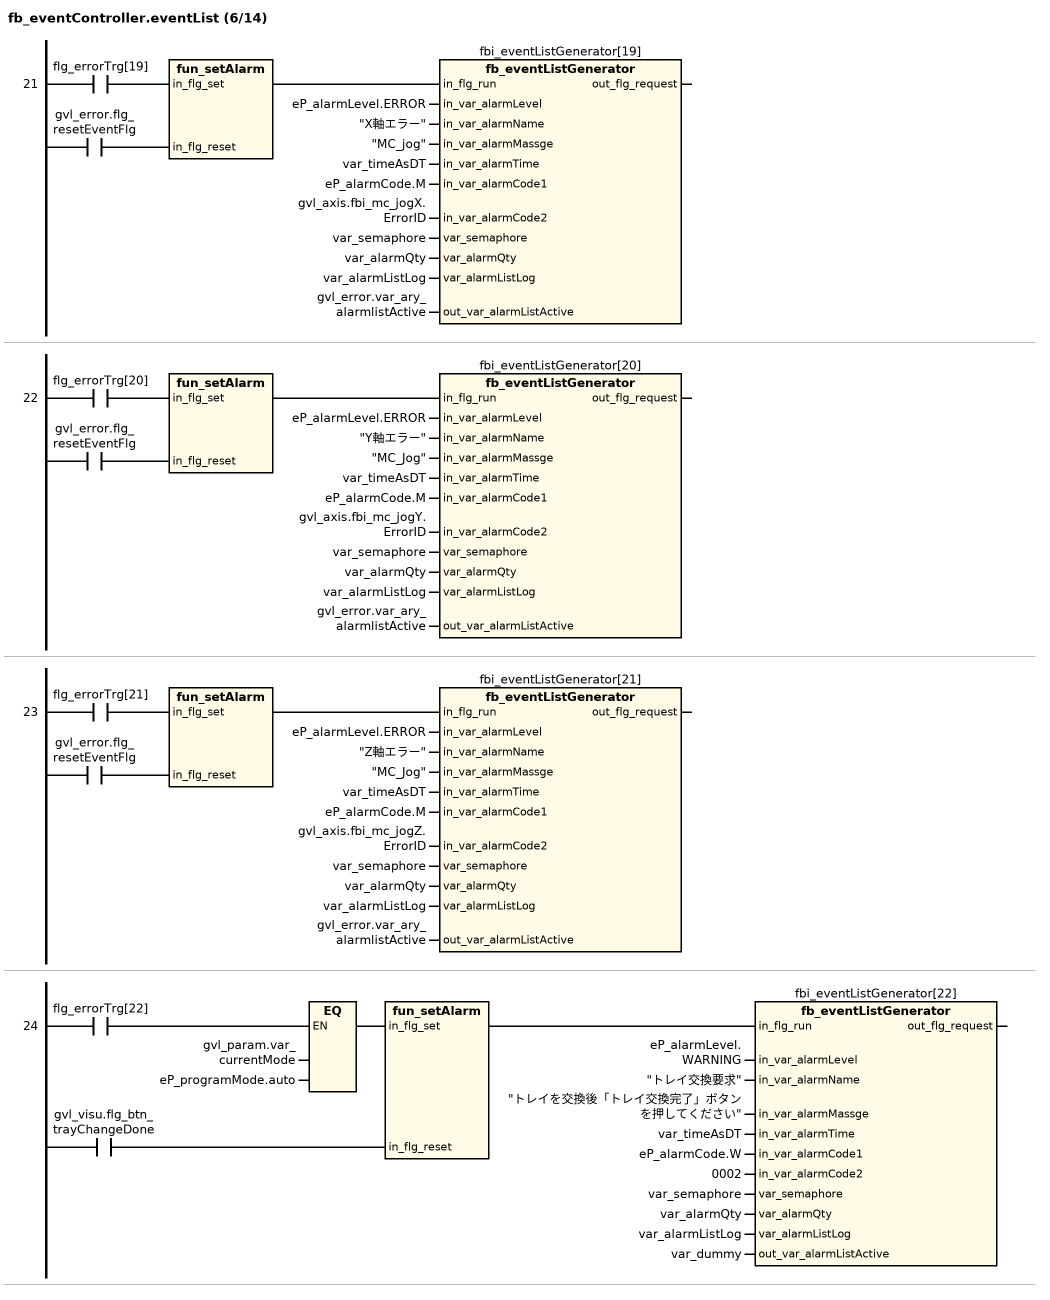
// NETWORK 21
fbi_eventListGenerator[19](
    in_flg_run := fun_setAlarm(in_flg_set := flg_errorTrg[19], in_flg_reset := gvl_error.flg_resetEventFlg),
    in_var_alarmLevel := eP_alarmLevel.ERROR,
    in_var_alarmName := "X軸エラー",
    in_var_alarmMassge := "MC_jog",
    in_var_alarmTime := var_timeAsDT,
    in_var_alarmCode1 := eP_alarmCode.M,
    in_var_alarmCode2 := gvl_axis.fbi_mc_jogX.ErrorID,
    var_semaphore := var_semaphore,
    var_alarmQty := var_alarmQty,
    var_alarmListLog := var_alarmListLog,
    out_var_alarmListActive := gvl_error.var_ary_alarmlistActive); // fb_eventListGenerator

// NETWORK 22
fbi_eventListGenerator[20](
    in_flg_run := fun_setAlarm(in_flg_set := flg_errorTrg[20], in_flg_reset := gvl_error.flg_resetEventFlg),
    in_var_alarmLevel := eP_alarmLevel.ERROR,
    in_var_alarmName := "Y軸エラー",
    in_var_alarmMassge := "MC_Jog",
    in_var_alarmTime := var_timeAsDT,
    in_var_alarmCode1 := eP_alarmCode.M,
    in_var_alarmCode2 := gvl_axis.fbi_mc_jogY.ErrorID,
    var_semaphore := var_semaphore,
    var_alarmQty := var_alarmQty,
    var_alarmListLog := var_alarmListLog,
    out_var_alarmListActive := gvl_error.var_ary_alarmlistActive); // fb_eventListGenerator

// NETWORK 23
fbi_eventListGenerator[21](
    in_flg_run := fun_setAlarm(in_flg_set := flg_errorTrg[21], in_flg_reset := gvl_error.flg_resetEventFlg),
    in_var_alarmLevel := eP_alarmLevel.ERROR,
    in_var_alarmName := "Z軸エラー",
    in_var_alarmMassge := "MC_Jog",
    in_var_alarmTime := var_timeAsDT,
    in_var_alarmCode1 := eP_alarmCode.M,
    in_var_alarmCode2 := gvl_axis.fbi_mc_jogZ.ErrorID,
    var_semaphore := var_semaphore,
    var_alarmQty := var_alarmQty,
    var_alarmListLog := var_alarmListLog,
    out_var_alarmListActive := gvl_error.var_ary_alarmlistActive); // fb_eventListGenerator

// NETWORK 24
fbi_eventListGenerator[22](
    in_flg_run := fun_setAlarm(in_flg_set := flg_errorTrg[22] AND gvl_param.var_currentMode = eP_programMode.auto, in_flg_reset := gvl_visu.flg_btn_trayChangeDone),
    in_var_alarmLevel := eP_alarmLevel.WARNING,
    in_var_alarmName := "トレイ交換要求",
    in_var_alarmMassge := "トレイを交換後「トレイ交換完了」ボタンを押してください",
    in_var_alarmTime := var_timeAsDT,
    in_var_alarmCode1 := eP_alarmCode.W,
    in_var_alarmCode2 := 0002,
    var_semaphore := var_semaphore,
    var_alarmQty := var_alarmQty,
    var_alarmListLog := var_alarmListLog,
    out_var_alarmListActive := var_dummy); // fb_eventListGenerator

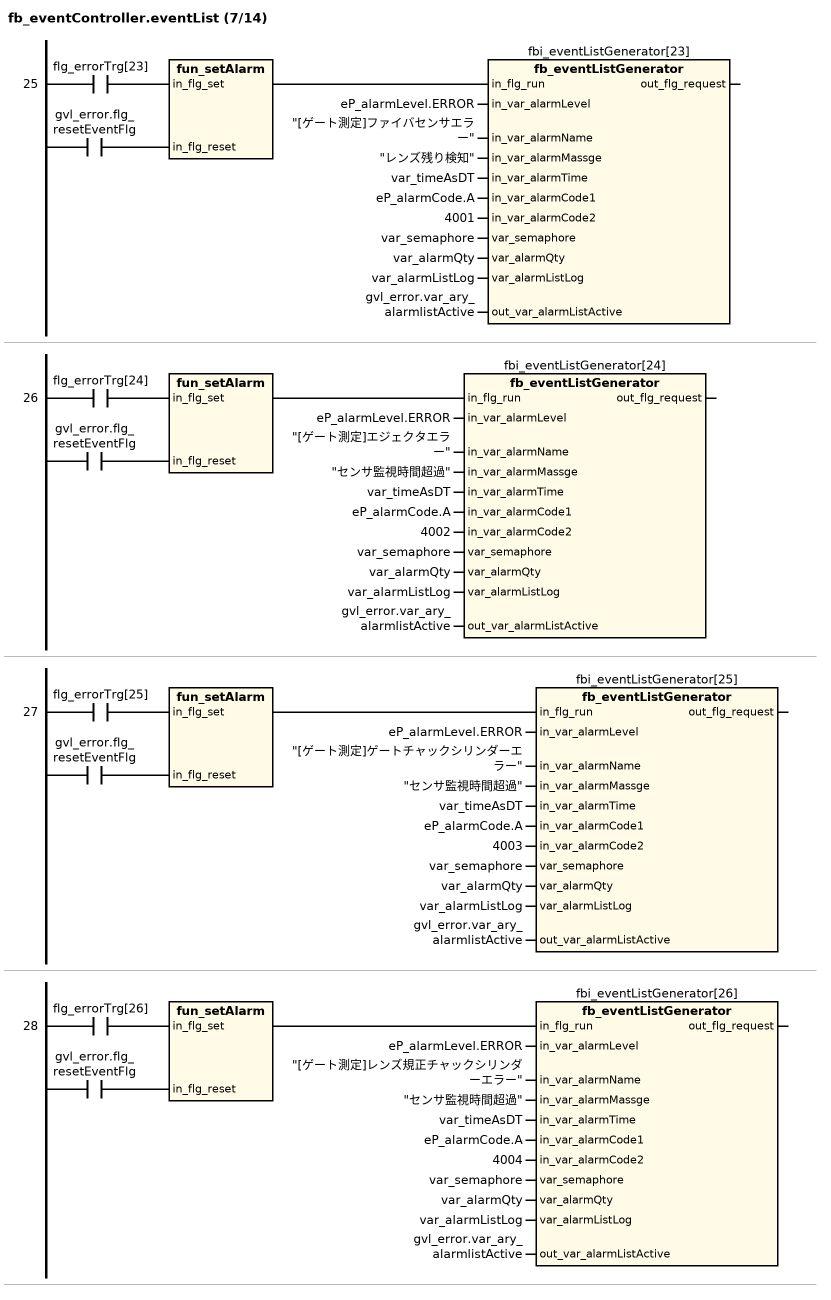
// NETWORK 25
fbi_eventListGenerator[23](
    in_flg_run := fun_setAlarm(in_flg_set := flg_errorTrg[23], in_flg_reset := gvl_error.flg_resetEventFlg),
    in_var_alarmLevel := eP_alarmLevel.ERROR,
    in_var_alarmName := "[ゲート測定]ファイバセンサエラー",
    in_var_alarmMassge := "レンズ残り検知",
    in_var_alarmTime := var_timeAsDT,
    in_var_alarmCode1 := eP_alarmCode.A,
    in_var_alarmCode2 := 4001,
    var_semaphore := var_semaphore,
    var_alarmQty := var_alarmQty,
    var_alarmListLog := var_alarmListLog,
    out_var_alarmListActive := gvl_error.var_ary_alarmlistActive); // fb_eventListGenerator

// NETWORK 26
fbi_eventListGenerator[24](
    in_flg_run := fun_setAlarm(in_flg_set := flg_errorTrg[24], in_flg_reset := gvl_error.flg_resetEventFlg),
    in_var_alarmLevel := eP_alarmLevel.ERROR,
    in_var_alarmName := "[ゲート測定]エジェクタエラー",
    in_var_alarmMassge := "センサ監視時間超過",
    in_var_alarmTime := var_timeAsDT,
    in_var_alarmCode1 := eP_alarmCode.A,
    in_var_alarmCode2 := 4002,
    var_semaphore := var_semaphore,
    var_alarmQty := var_alarmQty,
    var_alarmListLog := var_alarmListLog,
    out_var_alarmListActive := gvl_error.var_ary_alarmlistActive); // fb_eventListGenerator

// NETWORK 27
fbi_eventListGenerator[25](
    in_flg_run := fun_setAlarm(in_flg_set := flg_errorTrg[25], in_flg_reset := gvl_error.flg_resetEventFlg),
    in_var_alarmLevel := eP_alarmLevel.ERROR,
    in_var_alarmName := "[ゲート測定]ゲートチャックシリンダーエラー",
    in_var_alarmMassge := "センサ監視時間超過",
    in_var_alarmTime := var_timeAsDT,
    in_var_alarmCode1 := eP_alarmCode.A,
    in_var_alarmCode2 := 4003,
    var_semaphore := var_semaphore,
    var_alarmQty := var_alarmQty,
    var_alarmListLog := var_alarmListLog,
    out_var_alarmListActive := gvl_error.var_ary_alarmlistActive); // fb_eventListGenerator

// NETWORK 28
fbi_eventListGenerator[26](
    in_flg_run := fun_setAlarm(in_flg_set := flg_errorTrg[26], in_flg_reset := gvl_error.flg_resetEventFlg),
    in_var_alarmLevel := eP_alarmLevel.ERROR,
    in_var_alarmName := "[ゲート測定]レンズ規正チャックシリンダーエラー",
    in_var_alarmMassge := "センサ監視時間超過",
    in_var_alarmTime := var_timeAsDT,
    in_var_alarmCode1 := eP_alarmCode.A,
    in_var_alarmCode2 := 4004,
    var_semaphore := var_semaphore,
    var_alarmQty := var_alarmQty,
    var_alarmListLog := var_alarmListLog,
    out_var_alarmListActive := gvl_error.var_ary_alarmlistActive); // fb_eventListGenerator

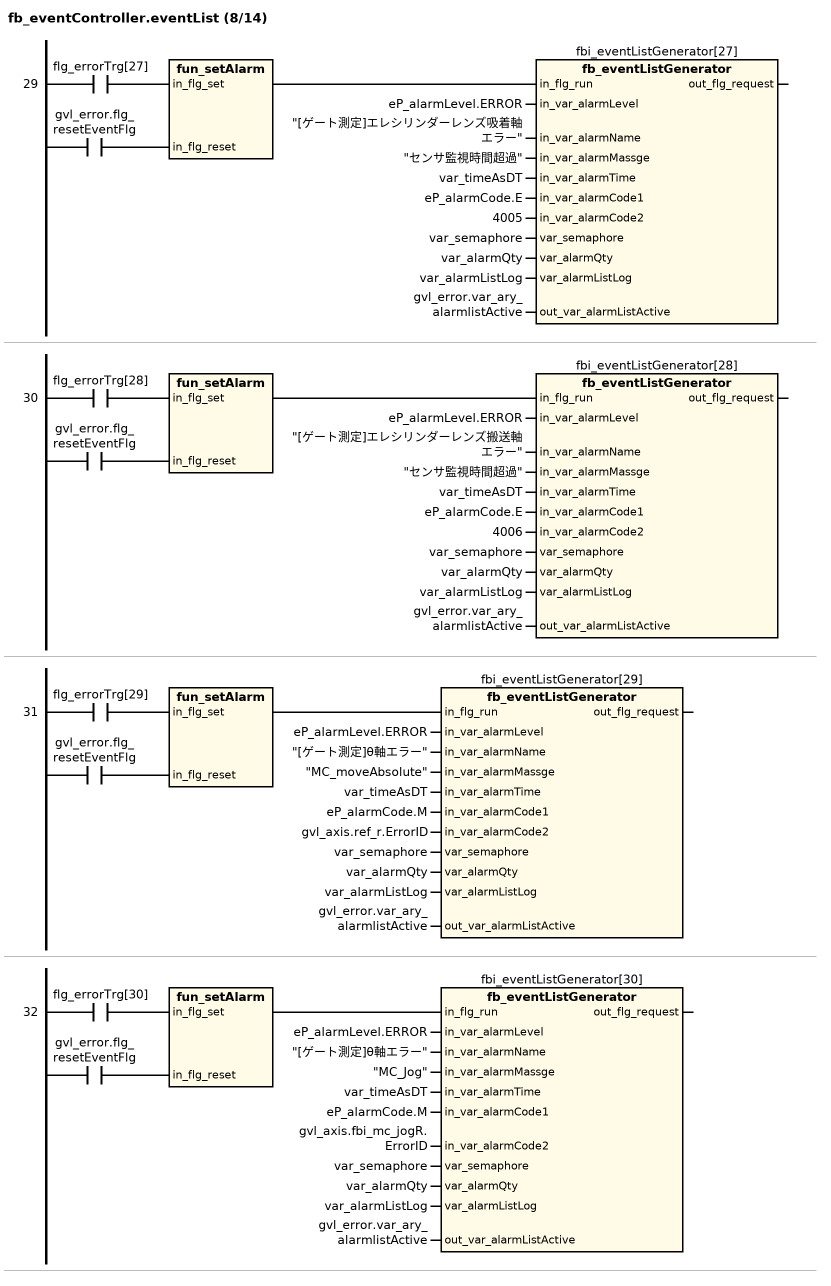
// NETWORK 29
fbi_eventListGenerator[27](
    in_flg_run := fun_setAlarm(in_flg_set := flg_errorTrg[27], in_flg_reset := gvl_error.flg_resetEventFlg),
    in_var_alarmLevel := eP_alarmLevel.ERROR,
    in_var_alarmName := "[ゲート測定]エレシリンダーレンズ吸着軸エラー",
    in_var_alarmMassge := "センサ監視時間超過",
    in_var_alarmTime := var_timeAsDT,
    in_var_alarmCode1 := eP_alarmCode.E,
    in_var_alarmCode2 := 4005,
    var_semaphore := var_semaphore,
    var_alarmQty := var_alarmQty,
    var_alarmListLog := var_alarmListLog,
    out_var_alarmListActive := gvl_error.var_ary_alarmlistActive); // fb_eventListGenerator

// NETWORK 30
fbi_eventListGenerator[28](
    in_flg_run := fun_setAlarm(in_flg_set := flg_errorTrg[28], in_flg_reset := gvl_error.flg_resetEventFlg),
    in_var_alarmLevel := eP_alarmLevel.ERROR,
    in_var_alarmName := "[ゲート測定]エレシリンダーレンズ搬送軸エラー",
    in_var_alarmMassge := "センサ監視時間超過",
    in_var_alarmTime := var_timeAsDT,
    in_var_alarmCode1 := eP_alarmCode.E,
    in_var_alarmCode2 := 4006,
    var_semaphore := var_semaphore,
    var_alarmQty := var_alarmQty,
    var_alarmListLog := var_alarmListLog,
    out_var_alarmListActive := gvl_error.var_ary_alarmlistActive); // fb_eventListGenerator

// NETWORK 31
fbi_eventListGenerator[29](
    in_flg_run := fun_setAlarm(in_flg_set := flg_errorTrg[29], in_flg_reset := gvl_error.flg_resetEventFlg),
    in_var_alarmLevel := eP_alarmLevel.ERROR,
    in_var_alarmName := "[ゲート測定]θ軸エラー",
    in_var_alarmMassge := "MC_moveAbsolute",
    in_var_alarmTime := var_timeAsDT,
    in_var_alarmCode1 := eP_alarmCode.M,
    in_var_alarmCode2 := gvl_axis.ref_r.ErrorID,
    var_semaphore := var_semaphore,
    var_alarmQty := var_alarmQty,
    var_alarmListLog := var_alarmListLog,
    out_var_alarmListActive := gvl_error.var_ary_alarmlistActive); // fb_eventListGenerator

// NETWORK 32
fbi_eventListGenerator[30](
    in_flg_run := fun_setAlarm(in_flg_set := flg_errorTrg[30], in_flg_reset := gvl_error.flg_resetEventFlg),
    in_var_alarmLevel := eP_alarmLevel.ERROR,
    in_var_alarmName := "[ゲート測定]θ軸エラー",
    in_var_alarmMassge := "MC_Jog",
    in_var_alarmTime := var_timeAsDT,
    in_var_alarmCode1 := eP_alarmCode.M,
    in_var_alarmCode2 := gvl_axis.fbi_mc_jogR.ErrorID,
    var_semaphore := var_semaphore,
    var_alarmQty := var_alarmQty,
    var_alarmListLog := var_alarmListLog,
    out_var_alarmListActive := gvl_error.var_ary_alarmlistActive); // fb_eventListGenerator

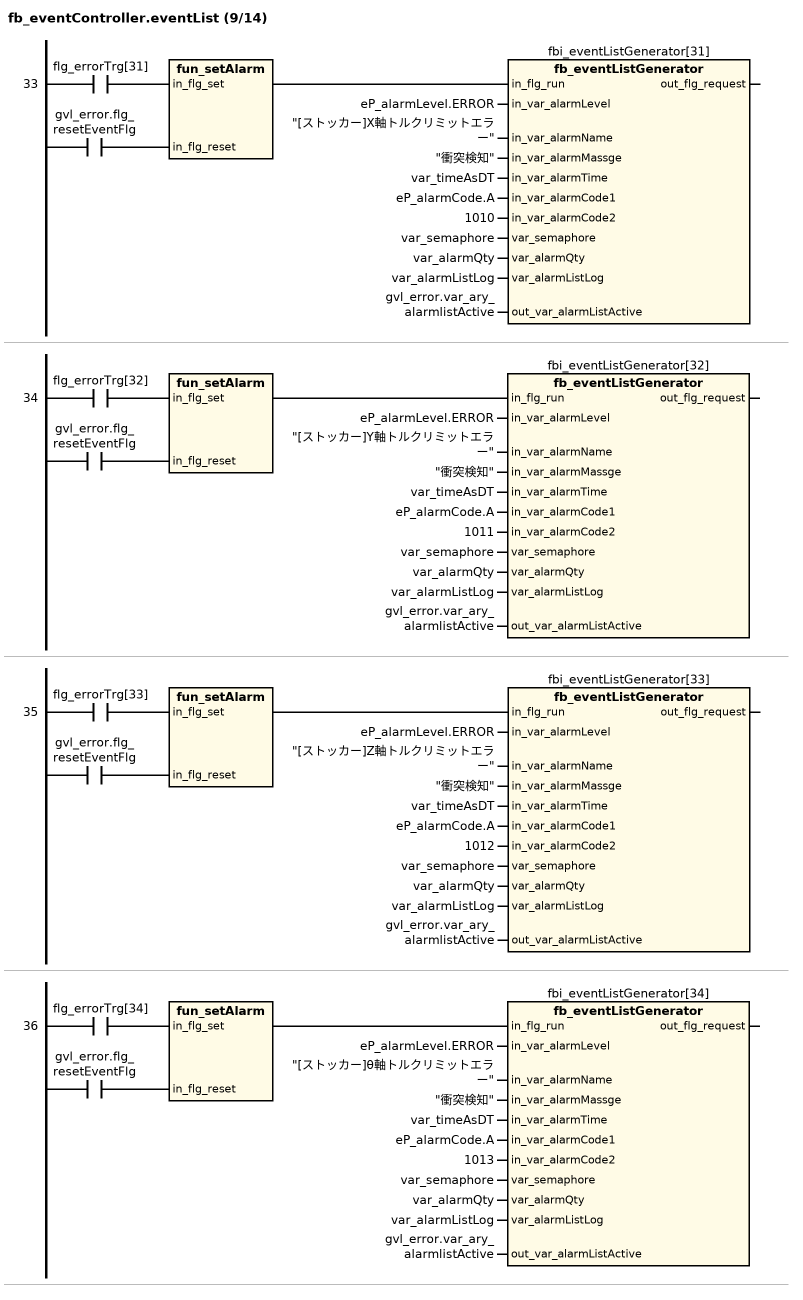
// NETWORK 33
fbi_eventListGenerator[31](
    in_flg_run := fun_setAlarm(in_flg_set := flg_errorTrg[31], in_flg_reset := gvl_error.flg_resetEventFlg),
    in_var_alarmLevel := eP_alarmLevel.ERROR,
    in_var_alarmName := "[ストッカー]X軸トルクリミットエラー",
    in_var_alarmMassge := "衝突検知",
    in_var_alarmTime := var_timeAsDT,
    in_var_alarmCode1 := eP_alarmCode.A,
    in_var_alarmCode2 := 1010,
    var_semaphore := var_semaphore,
    var_alarmQty := var_alarmQty,
    var_alarmListLog := var_alarmListLog,
    out_var_alarmListActive := gvl_error.var_ary_alarmlistActive); // fb_eventListGenerator

// NETWORK 34
fbi_eventListGenerator[32](
    in_flg_run := fun_setAlarm(in_flg_set := flg_errorTrg[32], in_flg_reset := gvl_error.flg_resetEventFlg),
    in_var_alarmLevel := eP_alarmLevel.ERROR,
    in_var_alarmName := "[ストッカー]Y軸トルクリミットエラー",
    in_var_alarmMassge := "衝突検知",
    in_var_alarmTime := var_timeAsDT,
    in_var_alarmCode1 := eP_alarmCode.A,
    in_var_alarmCode2 := 1011,
    var_semaphore := var_semaphore,
    var_alarmQty := var_alarmQty,
    var_alarmListLog := var_alarmListLog,
    out_var_alarmListActive := gvl_error.var_ary_alarmlistActive); // fb_eventListGenerator

// NETWORK 35
fbi_eventListGenerator[33](
    in_flg_run := fun_setAlarm(in_flg_set := flg_errorTrg[33], in_flg_reset := gvl_error.flg_resetEventFlg),
    in_var_alarmLevel := eP_alarmLevel.ERROR,
    in_var_alarmName := "[ストッカー]Z軸トルクリミットエラー",
    in_var_alarmMassge := "衝突検知",
    in_var_alarmTime := var_timeAsDT,
    in_var_alarmCode1 := eP_alarmCode.A,
    in_var_alarmCode2 := 1012,
    var_semaphore := var_semaphore,
    var_alarmQty := var_alarmQty,
    var_alarmListLog := var_alarmListLog,
    out_var_alarmListActive := gvl_error.var_ary_alarmlistActive); // fb_eventListGenerator

// NETWORK 36
fbi_eventListGenerator[34](
    in_flg_run := fun_setAlarm(in_flg_set := flg_errorTrg[34], in_flg_reset := gvl_error.flg_resetEventFlg),
    in_var_alarmLevel := eP_alarmLevel.ERROR,
    in_var_alarmName := "[ストッカー]θ軸トルクリミットエラー",
    in_var_alarmMassge := "衝突検知",
    in_var_alarmTime := var_timeAsDT,
    in_var_alarmCode1 := eP_alarmCode.A,
    in_var_alarmCode2 := 1013,
    var_semaphore := var_semaphore,
    var_alarmQty := var_alarmQty,
    var_alarmListLog := var_alarmListLog,
    out_var_alarmListActive := gvl_error.var_ary_alarmlistActive); // fb_eventListGenerator

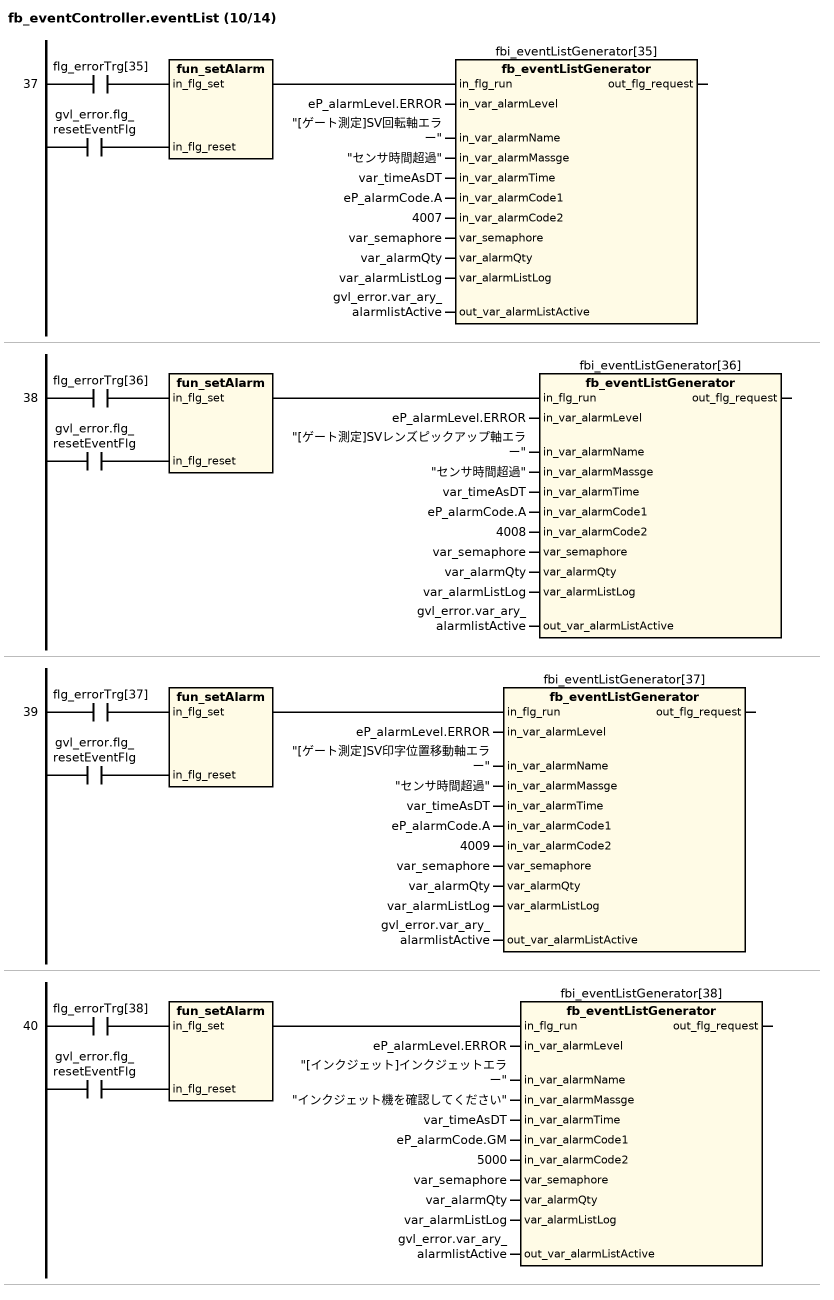
// NETWORK 37
fbi_eventListGenerator[35](
    in_flg_run := fun_setAlarm(in_flg_set := flg_errorTrg[35], in_flg_reset := gvl_error.flg_resetEventFlg),
    in_var_alarmLevel := eP_alarmLevel.ERROR,
    in_var_alarmName := "[ゲート測定]SV回転軸エラー",
    in_var_alarmMassge := "センサ時間超過",
    in_var_alarmTime := var_timeAsDT,
    in_var_alarmCode1 := eP_alarmCode.A,
    in_var_alarmCode2 := 4007,
    var_semaphore := var_semaphore,
    var_alarmQty := var_alarmQty,
    var_alarmListLog := var_alarmListLog,
    out_var_alarmListActive := gvl_error.var_ary_alarmlistActive); // fb_eventListGenerator

// NETWORK 38
fbi_eventListGenerator[36](
    in_flg_run := fun_setAlarm(in_flg_set := flg_errorTrg[36], in_flg_reset := gvl_error.flg_resetEventFlg),
    in_var_alarmLevel := eP_alarmLevel.ERROR,
    in_var_alarmName := "[ゲート測定]SVレンズピックアップ軸エラー",
    in_var_alarmMassge := "センサ時間超過",
    in_var_alarmTime := var_timeAsDT,
    in_var_alarmCode1 := eP_alarmCode.A,
    in_var_alarmCode2 := 4008,
    var_semaphore := var_semaphore,
    var_alarmQty := var_alarmQty,
    var_alarmListLog := var_alarmListLog,
    out_var_alarmListActive := gvl_error.var_ary_alarmlistActive); // fb_eventListGenerator

// NETWORK 39
fbi_eventListGenerator[37](
    in_flg_run := fun_setAlarm(in_flg_set := flg_errorTrg[37], in_flg_reset := gvl_error.flg_resetEventFlg),
    in_var_alarmLevel := eP_alarmLevel.ERROR,
    in_var_alarmName := "[ゲート測定]SV印字位置移動軸エラー",
    in_var_alarmMassge := "センサ時間超過",
    in_var_alarmTime := var_timeAsDT,
    in_var_alarmCode1 := eP_alarmCode.A,
    in_var_alarmCode2 := 4009,
    var_semaphore := var_semaphore,
    var_alarmQty := var_alarmQty,
    var_alarmListLog := var_alarmListLog,
    out_var_alarmListActive := gvl_error.var_ary_alarmlistActive); // fb_eventListGenerator

// NETWORK 40
fbi_eventListGenerator[38](
    in_flg_run := fun_setAlarm(in_flg_set := flg_errorTrg[38], in_flg_reset := gvl_error.flg_resetEventFlg),
    in_var_alarmLevel := eP_alarmLevel.ERROR,
    in_var_alarmName := "[インクジェット]インクジェットエラー",
    in_var_alarmMassge := "インクジェット機を確認してください",
    in_var_alarmTime := var_timeAsDT,
    in_var_alarmCode1 := eP_alarmCode.GM,
    in_var_alarmCode2 := 5000,
    var_semaphore := var_semaphore,
    var_alarmQty := var_alarmQty,
    var_alarmListLog := var_alarmListLog,
    out_var_alarmListActive := gvl_error.var_ary_alarmlistActive); // fb_eventListGenerator

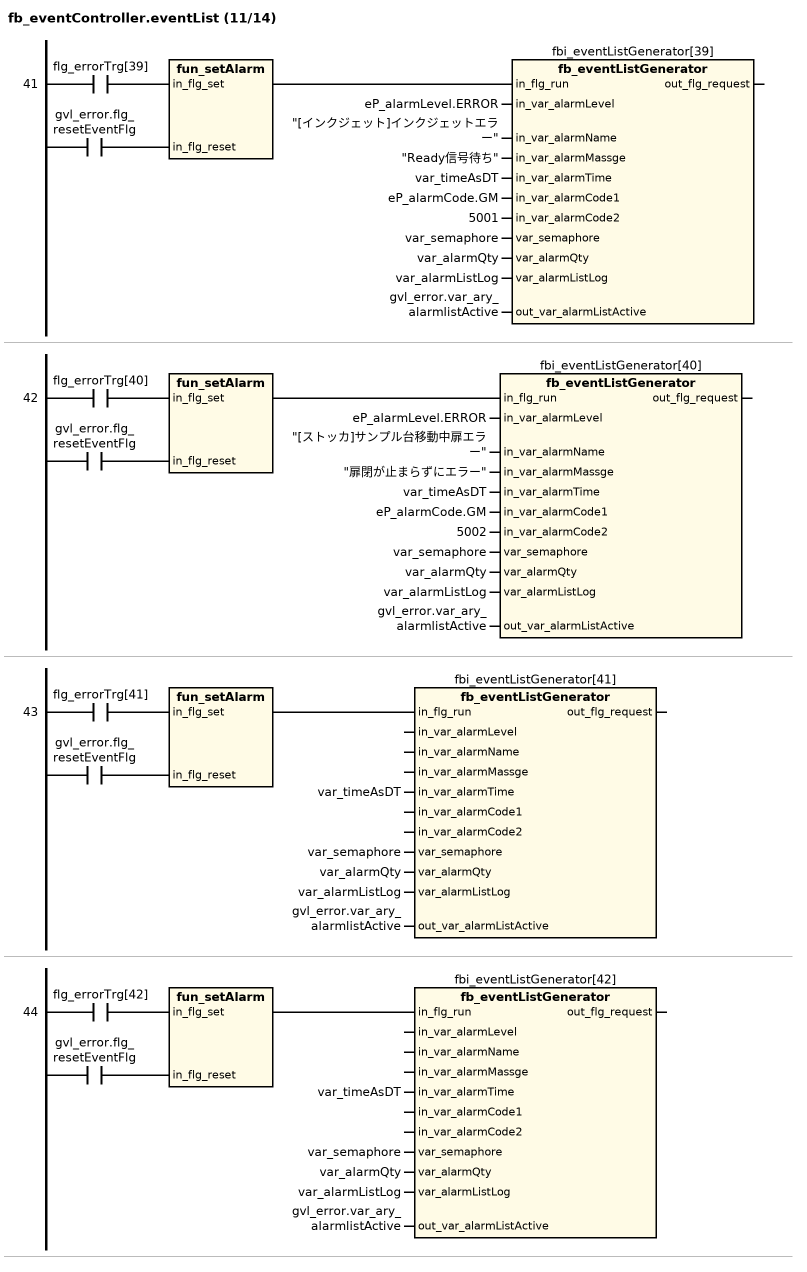
// NETWORK 41
fbi_eventListGenerator[39](
    in_flg_run := fun_setAlarm(in_flg_set := flg_errorTrg[39], in_flg_reset := gvl_error.flg_resetEventFlg),
    in_var_alarmLevel := eP_alarmLevel.ERROR,
    in_var_alarmName := "[インクジェット]インクジェットエラー",
    in_var_alarmMassge := "Ready信号待ち",
    in_var_alarmTime := var_timeAsDT,
    in_var_alarmCode1 := eP_alarmCode.GM,
    in_var_alarmCode2 := 5001,
    var_semaphore := var_semaphore,
    var_alarmQty := var_alarmQty,
    var_alarmListLog := var_alarmListLog,
    out_var_alarmListActive := gvl_error.var_ary_alarmlistActive); // fb_eventListGenerator

// NETWORK 42
fbi_eventListGenerator[40](
    in_flg_run := fun_setAlarm(in_flg_set := flg_errorTrg[40], in_flg_reset := gvl_error.flg_resetEventFlg),
    in_var_alarmLevel := eP_alarmLevel.ERROR,
    in_var_alarmName := "[ストッカ]サンプル台移動中扉エラー",
    in_var_alarmMassge := "扉閉が止まらずにエラー",
    in_var_alarmTime := var_timeAsDT,
    in_var_alarmCode1 := eP_alarmCode.GM,
    in_var_alarmCode2 := 5002,
    var_semaphore := var_semaphore,
    var_alarmQty := var_alarmQty,
    var_alarmListLog := var_alarmListLog,
    out_var_alarmListActive := gvl_error.var_ary_alarmlistActive); // fb_eventListGenerator

// NETWORK 43
fbi_eventListGenerator[41](
    in_flg_run := fun_setAlarm(in_flg_set := flg_errorTrg[41], in_flg_reset := gvl_error.flg_resetEventFlg),
    in_var_alarmTime := var_timeAsDT,
    var_semaphore := var_semaphore,
    var_alarmQty := var_alarmQty,
    var_alarmListLog := var_alarmListLog,
    out_var_alarmListActive := gvl_error.var_ary_alarmlistActive); // fb_eventListGenerator

// NETWORK 44
fbi_eventListGenerator[42](
    in_flg_run := fun_setAlarm(in_flg_set := flg_errorTrg[42], in_flg_reset := gvl_error.flg_resetEventFlg),
    in_var_alarmTime := var_timeAsDT,
    var_semaphore := var_semaphore,
    var_alarmQty := var_alarmQty,
    var_alarmListLog := var_alarmListLog,
    out_var_alarmListActive := gvl_error.var_ary_alarmlistActive); // fb_eventListGenerator

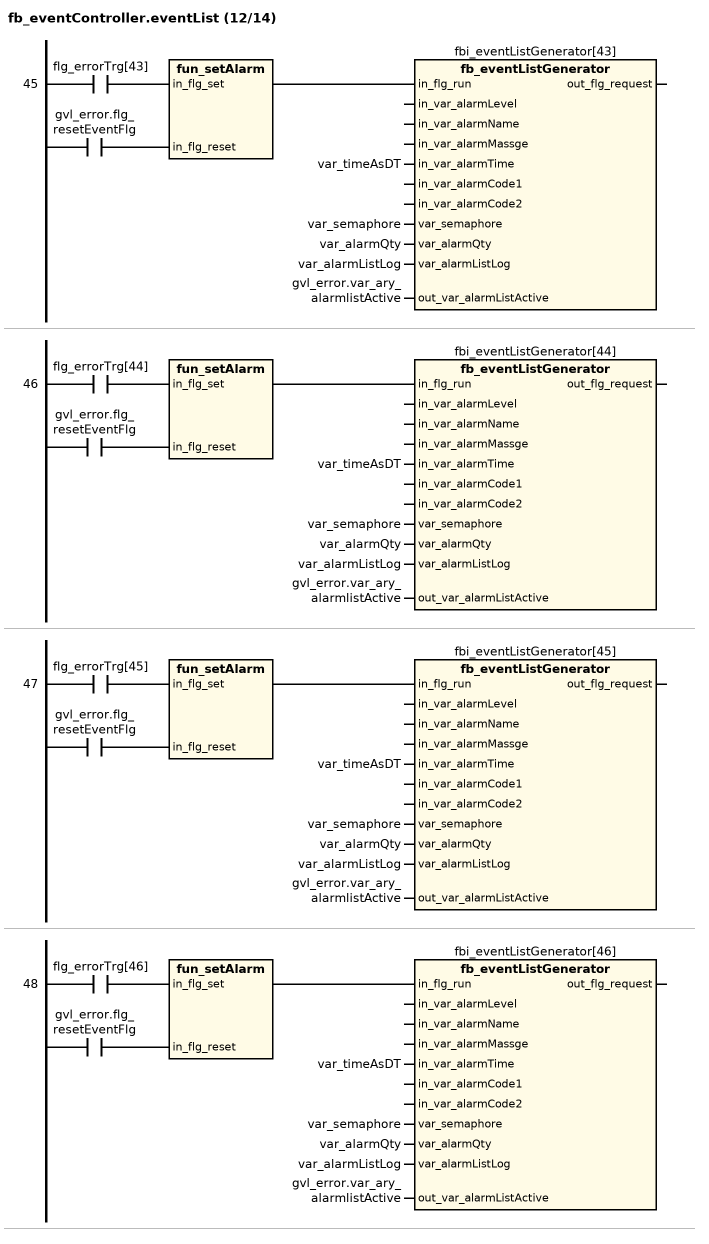
// NETWORK 45
fbi_eventListGenerator[43](
    in_flg_run := fun_setAlarm(in_flg_set := flg_errorTrg[43], in_flg_reset := gvl_error.flg_resetEventFlg),
    in_var_alarmTime := var_timeAsDT,
    var_semaphore := var_semaphore,
    var_alarmQty := var_alarmQty,
    var_alarmListLog := var_alarmListLog,
    out_var_alarmListActive := gvl_error.var_ary_alarmlistActive); // fb_eventListGenerator

// NETWORK 46
fbi_eventListGenerator[44](
    in_flg_run := fun_setAlarm(in_flg_set := flg_errorTrg[44], in_flg_reset := gvl_error.flg_resetEventFlg),
    in_var_alarmTime := var_timeAsDT,
    var_semaphore := var_semaphore,
    var_alarmQty := var_alarmQty,
    var_alarmListLog := var_alarmListLog,
    out_var_alarmListActive := gvl_error.var_ary_alarmlistActive); // fb_eventListGenerator

// NETWORK 47
fbi_eventListGenerator[45](
    in_flg_run := fun_setAlarm(in_flg_set := flg_errorTrg[45], in_flg_reset := gvl_error.flg_resetEventFlg),
    in_var_alarmTime := var_timeAsDT,
    var_semaphore := var_semaphore,
    var_alarmQty := var_alarmQty,
    var_alarmListLog := var_alarmListLog,
    out_var_alarmListActive := gvl_error.var_ary_alarmlistActive); // fb_eventListGenerator

// NETWORK 48
fbi_eventListGenerator[46](
    in_flg_run := fun_setAlarm(in_flg_set := flg_errorTrg[46], in_flg_reset := gvl_error.flg_resetEventFlg),
    in_var_alarmTime := var_timeAsDT,
    var_semaphore := var_semaphore,
    var_alarmQty := var_alarmQty,
    var_alarmListLog := var_alarmListLog,
    out_var_alarmListActive := gvl_error.var_ary_alarmlistActive); // fb_eventListGenerator

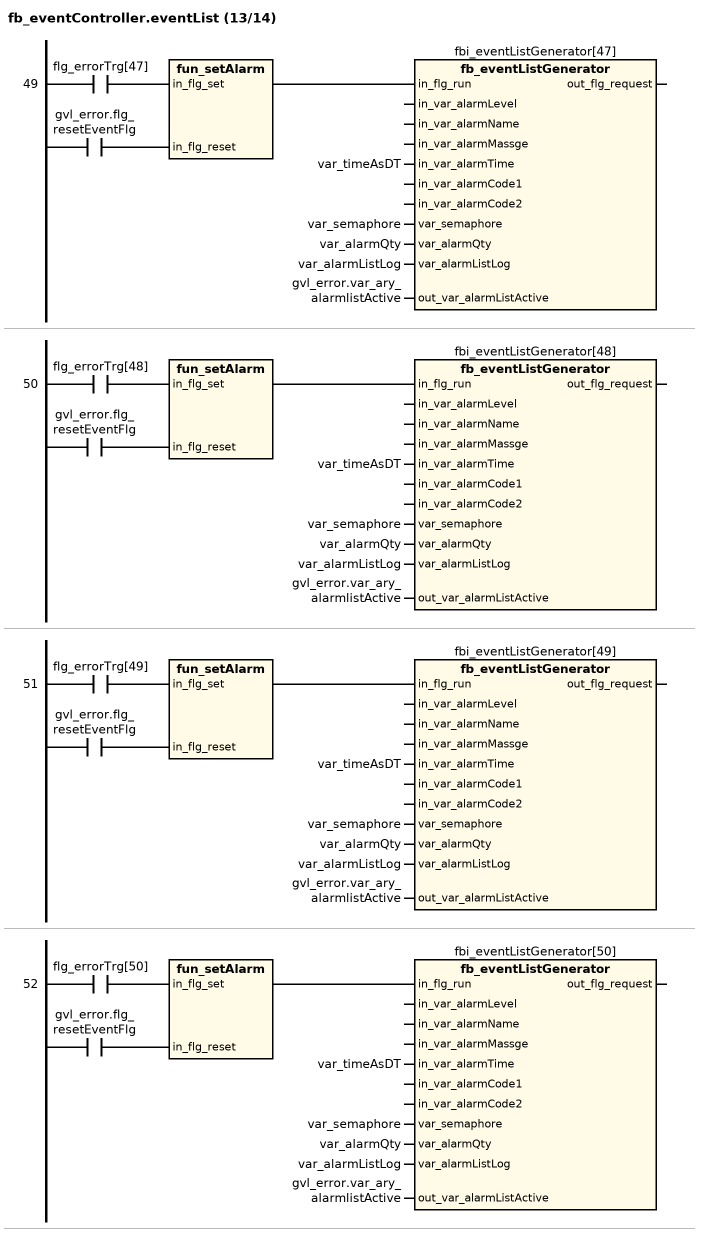
// NETWORK 49
fbi_eventListGenerator[47](
    in_flg_run := fun_setAlarm(in_flg_set := flg_errorTrg[47], in_flg_reset := gvl_error.flg_resetEventFlg),
    in_var_alarmTime := var_timeAsDT,
    var_semaphore := var_semaphore,
    var_alarmQty := var_alarmQty,
    var_alarmListLog := var_alarmListLog,
    out_var_alarmListActive := gvl_error.var_ary_alarmlistActive); // fb_eventListGenerator

// NETWORK 50
fbi_eventListGenerator[48](
    in_flg_run := fun_setAlarm(in_flg_set := flg_errorTrg[48], in_flg_reset := gvl_error.flg_resetEventFlg),
    in_var_alarmTime := var_timeAsDT,
    var_semaphore := var_semaphore,
    var_alarmQty := var_alarmQty,
    var_alarmListLog := var_alarmListLog,
    out_var_alarmListActive := gvl_error.var_ary_alarmlistActive); // fb_eventListGenerator

// NETWORK 51
fbi_eventListGenerator[49](
    in_flg_run := fun_setAlarm(in_flg_set := flg_errorTrg[49], in_flg_reset := gvl_error.flg_resetEventFlg),
    in_var_alarmTime := var_timeAsDT,
    var_semaphore := var_semaphore,
    var_alarmQty := var_alarmQty,
    var_alarmListLog := var_alarmListLog,
    out_var_alarmListActive := gvl_error.var_ary_alarmlistActive); // fb_eventListGenerator

// NETWORK 52
fbi_eventListGenerator[50](
    in_flg_run := fun_setAlarm(in_flg_set := flg_errorTrg[50], in_flg_reset := gvl_error.flg_resetEventFlg),
    in_var_alarmTime := var_timeAsDT,
    var_semaphore := var_semaphore,
    var_alarmQty := var_alarmQty,
    var_alarmListLog := var_alarmListLog,
    out_var_alarmListActive := gvl_error.var_ary_alarmlistActive); // fb_eventListGenerator

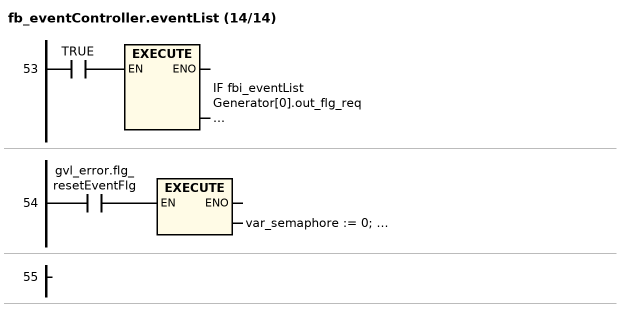
// NETWORK 53
IF fbi_eventListGenerator[0].out_flg_request OR
	fbi_eventListGenerator[1].out_flg_request OR
	fbi_eventListGenerator[2].out_flg_request OR
	fbi_eventListGenerator[3].out_flg_request OR
	fbi_eventListGenerator[4].out_flg_request OR
	fbi_eventListGenerator[5].out_flg_request OR
	fbi_eventListGenerator[6].out_flg_request OR
	fbi_eventListGenerator[7].out_flg_request OR
	fbi_eventListGenerator[8].out_flg_request OR
	fbi_eventListGenerator[9].out_flg_request OR
	fbi_eventListGenerator[10].out_flg_request OR
	fbi_eventListGenerator[11].out_flg_request OR
	fbi_eventListGenerator[12].out_flg_request OR
	fbi_eventListGenerator[13].out_flg_request OR
	fbi_eventListGenerator[14].out_flg_request OR
	fbi_eventListGenerator[15].out_flg_request OR
	fbi_eventListGenerator[16].out_flg_request OR
	fbi_eventListGenerator[17].out_flg_request OR
	fbi_eventListGenerator[18].out_flg_request OR
	fbi_eventListGenerator[19].out_flg_request OR
	fbi_eventListGenerator[20].out_flg_request OR
	fbi_eventListGenerator[21].out_flg_request OR
	fbi_eventListGenerator[22].out_flg_request OR
	fbi_eventListGenerator[23].out_flg_request OR
	fbi_eventListGenerator[24].out_flg_request OR
	fbi_eventListGenerator[25].out_flg_request OR
	fbi_eventListGenerator[26].out_flg_request OR
	fbi_eventListGenerator[27].out_flg_request OR
	fbi_eventListGenerator[28].out_flg_request OR
	fbi_eventListGenerator[29].out_flg_request OR
	fbi_eventListGenerator[30].out_flg_request OR
	fbi_eventListGenerator[31].out_flg_request OR
	fbi_eventListGenerator[32].out_flg_request OR
	fbi_eventListGenerator[33].out_flg_request OR
	fbi_eventListGenerator[34].out_flg_request OR
	fbi_eventListGenerator[35].out_flg_request OR
	fbi_eventListGenerator[36].out_flg_request OR
	fbi_eventListGenerator[37].out_flg_request OR
	fbi_eventListGenerator[38].out_flg_request OR
	fbi_eventListGenerator[39].out_flg_request OR
	fbi_eventListGenerator[40].out_flg_request OR
	fbi_eventListGenerator[41].out_flg_request OR
	fbi_eventListGenerator[42].out_flg_request OR
	fbi_eventListGenerator[43].out_flg_request OR
	fbi_eventListGenerator[44].out_flg_request OR
	fbi_eventListGenerator[44].out_flg_request OR
	fbi_eventListGenerator[45].out_flg_request OR
	fbi_eventListGenerator[46].out_flg_request OR
	fbi_eventListGenerator[47].out_flg_request OR
	fbi_eventListGenerator[48].out_flg_request OR
	fbi_eventListGenerator[49].out_flg_request OR
	fbi_eventListGenerator[50].out_flg_request THEN
		flg_reqUpdate := TRUE;
ELSE
	flg_reqUpdate := FALSE;
END_IF

// NETWORK 54
IF gvl_error.flg_resetEventFlg THEN
    var_semaphore := 0;
    var_alarmQty := 0;
END_IF

// NETWORK 55
END_ACTION

END_FUNCTION_BLOCK

// ---- FBs/error/fb_eventListGenerator.TcPOU
FUNCTION_BLOCK fb_eventListGenerator
VAR_INPUT
	in_flg_run : BOOL;
	in_var_alarmLevel : eP_alarmLevel;
	in_var_alarmName : WSTRING;
	in_var_alarmMassge : WSTRING;
	in_var_alarmTime : DT;
	in_var_alarmCode1 : eP_alarmCode;
	in_var_alarmCode2 : UDINT;
END_VAR
VAR_IN_OUT
	var_semaphore : INT;
	var_alarmQty : INT;
	var_alarmListLog: s_alarmList;
	out_var_alarmListActive:ARRAY[1..10] OF s_str_alarmList;
END_VAR
VAR_OUTPUT
	out_flg_request : BOOL;
END_VAR
VAR
	buf_var_alarmList : s_alarmList;
	buf_var_str_alarmList : s_str_alarmList;
	flg_active: BOOL;
	buf_var_semaphore: INT;
	var_process: INT;

	delayTimer: TON;
END_VAR

VAR_STAT
	flg_LvError : BOOL;
	flg_LvWarning : BOOL;
	flg_LvInfo : BOOL;
END_VAR
VAR // added by the converter: edge detectors and wires of the graphical bodies
    _rt1, _rt2, _rt3, _rt4 : R_TRIG;
    _w1, _w2, _w3, _w4, _w5 : BOOL;
    _ft1, _ft2 : F_TRIG;
END_VAR

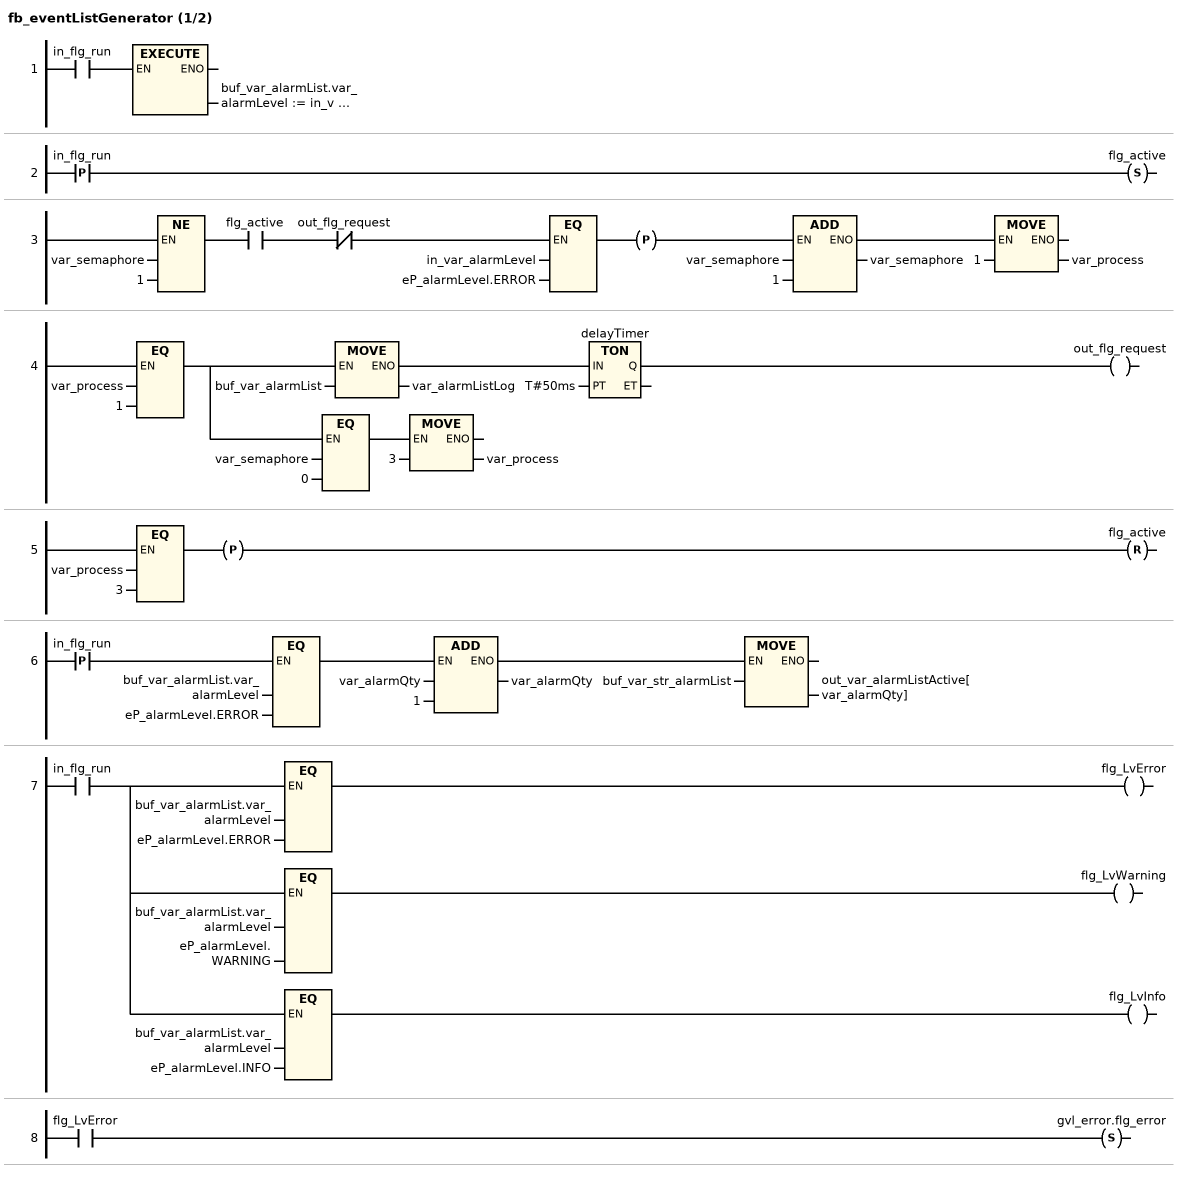
// NETWORK 1
IF in_flg_run THEN
    buf_var_alarmList.var_alarmLevel := in_var_alarmLevel;
    buf_var_alarmList.var_alarmName := in_var_alarmName;
    buf_var_alarmList.var_alarmMassge := in_var_alarmMassge;
    buf_var_alarmList.var_alarmTime := in_var_alarmTime;
    buf_var_alarmList.var_alarmCode1 := in_var_alarmCode1;
    buf_var_alarmList.var_alarmCode2 := in_var_alarmCode2;
    
    
    buf_var_str_alarmList.var_alarmName := in_var_alarmName;
    buf_var_str_alarmList.var_alarmMassge := in_var_alarmMassge;
    buf_var_str_alarmList.var_alarmTime := DT_TO_STRING(in_var_alarmTime);
    buf_var_str_alarmList.var_alarmCode1 := in_var_alarmCode1;
    buf_var_str_alarmList.var_alarmCode2 := UDINT_TO_STRING(in_var_alarmCode2);
END_IF

// NETWORK 2
_rt1(CLK := in_flg_run);
flg_active S= _rt1.Q;

// NETWORK 3
_rt2(CLK := var_semaphore <> 1 AND flg_active AND NOT out_flg_request AND in_var_alarmLevel = eP_alarmLevel.ERROR);
_w1 := _rt2.Q;
IF _w1 THEN var_semaphore := var_semaphore + 1; END_IF
IF _w1 THEN var_process := 1; END_IF

// NETWORK 4
_w2 := var_process = 1;
IF _w2 THEN var_alarmListLog := buf_var_alarmList; END_IF
delayTimer(IN := _w2, PT := T#50ms); // TON
out_flg_request := delayTimer.Q;
IF _w2 AND var_semaphore = 0 THEN var_process := 3; END_IF

// NETWORK 5
_rt3(CLK := var_process = 3);
flg_active R= _rt3.Q;

// NETWORK 6
_rt4(CLK := in_flg_run);
_w3 := _rt4.Q AND buf_var_alarmList.var_alarmLevel = eP_alarmLevel.ERROR;
IF _w3 THEN var_alarmQty := var_alarmQty + 1; END_IF
IF _w3 THEN out_var_alarmListActive[var_alarmQty] := buf_var_str_alarmList; END_IF

// NETWORK 7
flg_LvError := in_flg_run AND buf_var_alarmList.var_alarmLevel = eP_alarmLevel.ERROR;
flg_LvWarning := in_flg_run AND buf_var_alarmList.var_alarmLevel = eP_alarmLevel.WARNING;
flg_LvInfo := in_flg_run AND buf_var_alarmList.var_alarmLevel = eP_alarmLevel.INFO;

// NETWORK 8
gvl_error.flg_error S= flg_LvError;

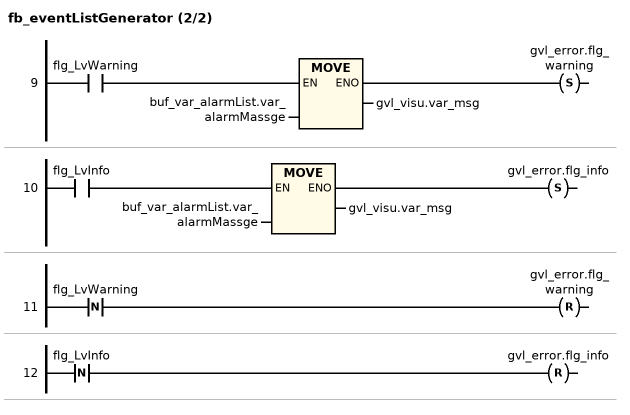
// NETWORK 9
_w4 := flg_LvWarning;
IF _w4 THEN gvl_visu.var_msg := buf_var_alarmList.var_alarmMassge; END_IF
gvl_error.flg_warning S= _w4;

// NETWORK 10
_w5 := flg_LvInfo;
IF _w5 THEN gvl_visu.var_msg := buf_var_alarmList.var_alarmMassge; END_IF
gvl_error.flg_info S= _w5;

// NETWORK 11
_ft1(CLK := flg_LvWarning);
gvl_error.flg_warning R= _ft1.Q;

// NETWORK 12
_ft2(CLK := flg_LvInfo);
gvl_error.flg_info R= _ft2.Q;

END_FUNCTION_BLOCK

// ---- FBs/error/fb_buzzerGenerater.TcPOU
FUNCTION_BLOCK fb_buzzerGenerater
VAR_INPUT
	in_flg_LvError : BOOL;
	in_flg_LvWarning : BOOL;
	in_flg_LvInfo : BOOL;
END_VAR
VAR_OUTPUT
	out_flg_buzzer : BOOL;
	out_flg_Yellow: BOOL;
END_VAR
VAR
	onDelay: TON;
	var_loop: INT;
	offDelay: TON;
	flg_buzzer_info: BOOL;
	flg_buzzer_warning: BOOL;
	flg_Yellow_warning: BOOL;
	flg_Yellow_manual: BOOL;
	flg_buzzer_error: BOOL;
END_VAR
VAR // added by the converter: edge detectors and wires of the graphical bodies
    _w1, _w2, _w3, _w4 : BOOL;
END_VAR

IF in_flg_LvError THEN
	flg_buzzer_error := TRUE;
ELSIF in_flg_LvWarning AND in_flg_LvError = FALSE THEN
	lv_warning();
ELSIF in_flg_LvInfo THEN
	//lv_info();
ELSE
	flg_Yellow_warning :=FALSE;
	flg_buzzer_warning := FALSE;
	flg_buzzer_error := FALSE;
END_IF

indicator();
manual();

ACTION indicator:
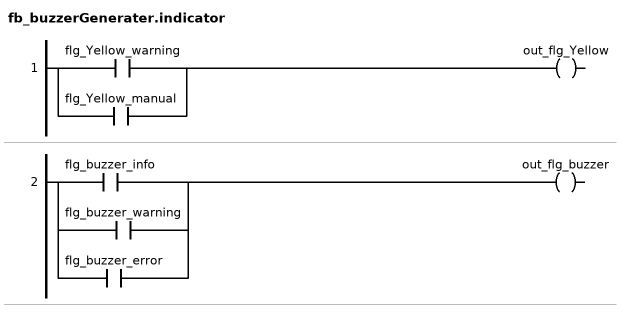
// NETWORK 1
out_flg_Yellow := flg_Yellow_warning OR flg_Yellow_manual;

// NETWORK 2
out_flg_buzzer := flg_buzzer_info OR flg_buzzer_warning OR flg_buzzer_error;
END_ACTION

ACTION lv_info:
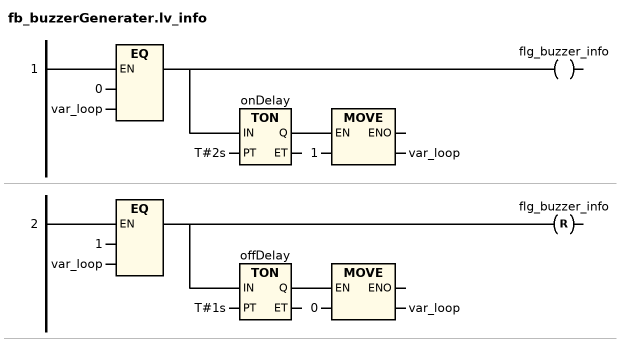
// NETWORK 1
_w1 := 0 = var_loop;
flg_buzzer_info := _w1;
onDelay(IN := _w1, PT := T#2s); // TON
IF onDelay.Q THEN var_loop := 1; END_IF

// NETWORK 2
_w2 := 1 = var_loop;
flg_buzzer_info R= _w2;
offDelay(IN := _w2, PT := T#1s); // TON
IF offDelay.Q THEN var_loop := 0; END_IF
END_ACTION

ACTION lv_warning:
